    stNO_LENS[885].fEnergy := 29760.957445; stNO_LENS[885].fLow := 4.726807; stNO_LENS[885].fHigh := 9.548423;
    stNO_LENS[886].fEnergy := 29820.538922; stNO_LENS[886].fLow := 4.709276; stNO_LENS[886].fHigh := 9.507957;
    stNO_LENS[887].fEnergy := 29880.239680; stNO_LENS[887].fLow := 4.691804; stNO_LENS[887].fHigh := 9.467684;
    stNO_LENS[888].fEnergy := 29940.059960; stNO_LENS[888].fLow := 4.674389; stNO_LENS[888].fHigh := 9.427603;
    stNO_LENS[889].fEnergy := 30000.000000; stNO_LENS[889].fLow := 4.657032; stNO_LENS[889].fHigh := 9.387713;
    stNO_LENS[890].fEnergy := 30068.760232; stNO_LENS[890].fLow := 4.637235; stNO_LENS[890].fHigh := 9.342285;
    stNO_LENS[891].fEnergy := 30128.957930; stNO_LENS[891].fLow := 4.620001; stNO_LENS[891].fHigh := 9.302803;
    stNO_LENS[892].fEnergy := 30189.276144; stNO_LENS[892].fLow := 4.602825; stNO_LENS[892].fHigh := 9.263510;
    stNO_LENS[893].fEnergy := 30249.715115; stNO_LENS[893].fLow := 4.585705; stNO_LENS[893].fHigh := 9.224405;
    stNO_LENS[894].fEnergy := 30310.275085; stNO_LENS[894].fLow := 4.568643; stNO_LENS[894].fHigh := 9.185487;
    stNO_LENS[895].fEnergy := 30370.956297; stNO_LENS[895].fLow := 4.551636; stNO_LENS[895].fHigh := 9.146757;
    stNO_LENS[896].fEnergy := 30431.758992; stNO_LENS[896].fLow := 4.534686; stNO_LENS[896].fHigh := 9.108213;
    stNO_LENS[897].fEnergy := 30492.683414; stNO_LENS[897].fLow := 4.517791; stNO_LENS[897].fHigh := 9.069854;
    stNO_LENS[898].fEnergy := 30553.729807; stNO_LENS[898].fLow := 4.500952; stNO_LENS[898].fHigh := 9.031681;
    stNO_LENS[899].fEnergy := 30614.898414; stNO_LENS[899].fLow := 4.484169; stNO_LENS[899].fHigh := 8.993692;
    stNO_LENS[900].fEnergy := 30676.189482; stNO_LENS[900].fLow := 4.467441; stNO_LENS[900].fHigh := 8.955886;
    stNO_LENS[901].fEnergy := 30737.603254; stNO_LENS[901].fLow := 4.450767; stNO_LENS[901].fHigh := 8.918263;
    stNO_LENS[902].fEnergy := 30799.139977; stNO_LENS[902].fLow := 4.434149; stNO_LENS[902].fHigh := 8.880822;
    stNO_LENS[903].fEnergy := 30860.799896; stNO_LENS[903].fLow := 4.417585; stNO_LENS[903].fHigh := 8.843563;
    stNO_LENS[904].fEnergy := 30922.583259; stNO_LENS[904].fLow := 4.401076; stNO_LENS[904].fHigh := 8.806484;
    stNO_LENS[905].fEnergy := 30984.490312; stNO_LENS[905].fLow := 4.384620; stNO_LENS[905].fHigh := 8.769586;
    stNO_LENS[906].fEnergy := 31046.521303; stNO_LENS[906].fLow := 4.368218; stNO_LENS[906].fHigh := 8.732867;
    stNO_LENS[907].fEnergy := 31108.676480; stNO_LENS[907].fLow := 4.351870; stNO_LENS[907].fHigh := 8.696327;
    stNO_LENS[908].fEnergy := 31170.956091; stNO_LENS[908].fLow := 4.335576; stNO_LENS[908].fHigh := 8.659965;
    stNO_LENS[909].fEnergy := 31233.360387; stNO_LENS[909].fLow := 4.319334; stNO_LENS[909].fHigh := 8.623781;
    stNO_LENS[910].fEnergy := 31295.889616; stNO_LENS[910].fLow := 4.303146; stNO_LENS[910].fHigh := 8.587773;
    stNO_LENS[911].fEnergy := 31358.544029; stNO_LENS[911].fLow := 4.287010; stNO_LENS[911].fHigh := 8.551941;
    stNO_LENS[912].fEnergy := 31421.323876; stNO_LENS[912].fLow := 4.270927; stNO_LENS[912].fHigh := 8.516285;
    stNO_LENS[913].fEnergy := 31484.229408; stNO_LENS[913].fLow := 4.254897; stNO_LENS[913].fHigh := 8.480803;
    stNO_LENS[914].fEnergy := 31547.260878; stNO_LENS[914].fLow := 4.238918; stNO_LENS[914].fHigh := 8.445496;
    stNO_LENS[915].fEnergy := 31610.418536; stNO_LENS[915].fLow := 4.222991; stNO_LENS[915].fHigh := 8.410362;
    stNO_LENS[916].fEnergy := 31673.702636; stNO_LENS[916].fLow := 4.207116; stNO_LENS[916].fHigh := 8.375401;
    stNO_LENS[917].fEnergy := 31737.113431; stNO_LENS[917].fLow := 4.191293; stNO_LENS[917].fHigh := 8.340611;
    stNO_LENS[918].fEnergy := 31800.651174; stNO_LENS[918].fLow := 4.175521; stNO_LENS[918].fHigh := 8.305993;
    stNO_LENS[919].fEnergy := 31864.316120; stNO_LENS[919].fLow := 4.159799; stNO_LENS[919].fHigh := 8.271546;
    stNO_LENS[920].fEnergy := 31928.108524; stNO_LENS[920].fLow := 4.144129; stNO_LENS[920].fHigh := 8.237269;
    stNO_LENS[921].fEnergy := 31992.028640; stNO_LENS[921].fLow := 4.128510; stNO_LENS[921].fHigh := 8.203161;
    stNO_LENS[922].fEnergy := 32056.076724; stNO_LENS[922].fLow := 4.112940; stNO_LENS[922].fHigh := 8.169222;
    stNO_LENS[923].fEnergy := 32120.253032; stNO_LENS[923].fLow := 4.097421; stNO_LENS[923].fHigh := 8.135452;
    stNO_LENS[924].fEnergy := 32184.557822; stNO_LENS[924].fLow := 4.081953; stNO_LENS[924].fHigh := 8.101848;
    stNO_LENS[925].fEnergy := 32248.991349; stNO_LENS[925].fLow := 4.066534; stNO_LENS[925].fHigh := 8.068411;
    stNO_LENS[926].fEnergy := 32313.553873; stNO_LENS[926].fLow := 4.051164; stNO_LENS[926].fHigh := 8.035141;
    stNO_LENS[927].fEnergy := 32378.245651; stNO_LENS[927].fLow := 4.035844; stNO_LENS[927].fHigh := 8.002035;
    stNO_LENS[928].fEnergy := 32443.066942; stNO_LENS[928].fLow := 4.020574; stNO_LENS[928].fHigh := 7.969095;
    stNO_LENS[929].fEnergy := 32508.018005; stNO_LENS[929].fLow := 4.005352; stNO_LENS[929].fHigh := 7.936319;
    stNO_LENS[930].fEnergy := 32573.099101; stNO_LENS[930].fLow := 3.990180; stNO_LENS[930].fHigh := 7.903706;
    stNO_LENS[931].fEnergy := 32638.310488; stNO_LENS[931].fLow := 3.975056; stNO_LENS[931].fHigh := 7.871256;
    stNO_LENS[932].fEnergy := 32703.652430; stNO_LENS[932].fLow := 3.959980; stNO_LENS[932].fHigh := 7.838968;
    stNO_LENS[933].fEnergy := 32769.125185; stNO_LENS[933].fLow := 3.944953; stNO_LENS[933].fHigh := 7.806842;
    stNO_LENS[934].fEnergy := 32834.729018; stNO_LENS[934].fLow := 3.929974; stNO_LENS[934].fHigh := 7.774876;
    stNO_LENS[935].fEnergy := 32900.464189; stNO_LENS[935].fLow := 3.915043; stNO_LENS[935].fHigh := 7.743071;
    stNO_LENS[936].fEnergy := 32966.330962; stNO_LENS[936].fLow := 3.900159; stNO_LENS[936].fHigh := 7.711425;
    stNO_LENS[937].fEnergy := 33032.329601; stNO_LENS[937].fLow := 3.885323; stNO_LENS[937].fHigh := 7.679938;
    stNO_LENS[938].fEnergy := 33098.460369; stNO_LENS[938].fLow := 3.870535; stNO_LENS[938].fHigh := 7.648610;
    stNO_LENS[939].fEnergy := 33164.723530; stNO_LENS[939].fLow := 3.855793; stNO_LENS[939].fHigh := 7.617439;
    stNO_LENS[940].fEnergy := 33231.119351; stNO_LENS[940].fLow := 3.841099; stNO_LENS[940].fHigh := 7.586425;
    stNO_LENS[941].fEnergy := 33297.648096; stNO_LENS[941].fLow := 3.826451; stNO_LENS[941].fHigh := 7.555568;
    stNO_LENS[942].fEnergy := 33364.310032; stNO_LENS[942].fLow := 3.811850; stNO_LENS[942].fHigh := 7.524866;
    stNO_LENS[943].fEnergy := 33431.105426; stNO_LENS[943].fLow := 3.797296; stNO_LENS[943].fHigh := 7.494320;
    stNO_LENS[944].fEnergy := 33498.034543; stNO_LENS[944].fLow := 3.782787; stNO_LENS[944].fHigh := 7.463928;
    stNO_LENS[945].fEnergy := 33565.097653; stNO_LENS[945].fLow := 3.768325; stNO_LENS[945].fHigh := 7.433689;
    stNO_LENS[946].fEnergy := 33632.295023; stNO_LENS[946].fLow := 3.753909; stNO_LENS[946].fHigh := 7.389056;
    stNO_LENS[947].fEnergy := 33699.626923; stNO_LENS[947].fLow := 3.739538; stNO_LENS[947].fHigh := 7.389056;
    stNO_LENS[948].fEnergy := 33767.093621; stNO_LENS[948].fLow := 3.725213; stNO_LENS[948].fHigh := 7.320540;
    stNO_LENS[949].fEnergy := 33834.695387; stNO_LENS[949].fLow := 3.710933; stNO_LENS[949].fHigh := 7.130147;
    stNO_LENS[950].fEnergy := 33902.432493; stNO_LENS[950].fLow := 3.696699; stNO_LENS[950].fHigh := 6.944706;
    stNO_LENS[951].fEnergy := 33970.305208; stNO_LENS[951].fLow := 3.682509; stNO_LENS[951].fHigh := 6.764088;
    stNO_LENS[952].fEnergy := 34038.313804; stNO_LENS[952].fLow := 3.668365; stNO_LENS[952].fHigh := 6.588167;
    stNO_LENS[953].fEnergy := 34106.458554; stNO_LENS[953].fLow := 3.654265; stNO_LENS[953].fHigh := 6.416822;
    stNO_LENS[954].fEnergy := 34174.739729; stNO_LENS[954].fLow := 3.640209; stNO_LENS[954].fHigh := 6.249933;
    stNO_LENS[955].fEnergy := 34243.157604; stNO_LENS[955].fLow := 3.626198; stNO_LENS[955].fHigh := 6.087384;
    stNO_LENS[956].fEnergy := 34311.712451; stNO_LENS[956].fLow := 3.612231; stNO_LENS[956].fHigh := 5.929063;
    stNO_LENS[957].fEnergy := 34380.404545; stNO_LENS[957].fLow := 3.598308; stNO_LENS[957].fHigh := 5.774860;
    stNO_LENS[958].fEnergy := 34449.234161; stNO_LENS[958].fLow := 3.584429; stNO_LENS[958].fHigh := 5.624667;
    stNO_LENS[959].fEnergy := 34518.201574; stNO_LENS[959].fLow := 3.570593; stNO_LENS[959].fHigh := 5.478381;
    stNO_LENS[960].fEnergy := 34587.307059; stNO_LENS[960].fLow := 3.556802; stNO_LENS[960].fHigh := 5.335899;
    stNO_LENS[961].fEnergy := 34656.550894; stNO_LENS[961].fLow := 3.543053; stNO_LENS[961].fHigh := 5.197123;
    stNO_LENS[962].fEnergy := 34725.933355; stNO_LENS[962].fLow := 3.529348; stNO_LENS[962].fHigh := 5.061956;
    stNO_LENS[963].fEnergy := 34795.454720; stNO_LENS[963].fLow := 3.515685; stNO_LENS[963].fHigh := 4.930304;
    stNO_LENS[964].fEnergy := 34865.115267; stNO_LENS[964].fLow := 3.502066; stNO_LENS[964].fHigh := 4.802077;
    stNO_LENS[965].fEnergy := 34934.915274; stNO_LENS[965].fLow := 3.488489; stNO_LENS[965].fHigh := 4.677184;
    stNO_LENS[966].fEnergy := 35004.855021; stNO_LENS[966].fLow := 3.474955; stNO_LENS[966].fHigh := 4.555540;
    stNO_LENS[967].fEnergy := 35074.934788; stNO_LENS[967].fLow := 3.461463; stNO_LENS[967].fHigh := 4.437059;
    stNO_LENS[968].fEnergy := 35145.154854; stNO_LENS[968].fLow := 3.448013; stNO_LENS[968].fHigh := 4.321660;
    stNO_LENS[969].fEnergy := 35215.515501; stNO_LENS[969].fLow := 3.434605; stNO_LENS[969].fHigh := 4.209262;
    stNO_LENS[970].fEnergy := 35286.017010; stNO_LENS[970].fLow := 3.421240; stNO_LENS[970].fHigh := 4.099787;
    stNO_LENS[971].fEnergy := 35356.659663; stNO_LENS[971].fLow := 3.407916; stNO_LENS[971].fHigh := 3.993160;
    stNO_LENS[972].fEnergy := 35427.443743; stNO_LENS[972].fLow := 3.394634; stNO_LENS[972].fHigh := 3.889306;
    stNO_LENS[973].fEnergy := 35498.369532; stNO_LENS[973].fLow := 3.381393; stNO_LENS[973].fHigh := 3.788152;
    stNO_LENS[974].fEnergy := 35569.437315; stNO_LENS[974].fLow := 3.368193; stNO_LENS[974].fHigh := 3.689630;
    stNO_LENS[975].fEnergy := 35640.647376; stNO_LENS[975].fLow := 3.355035; stNO_LENS[975].fHigh := 3.593670;
    stNO_LENS[976].fEnergy := 35712.000000; stNO_LENS[976].fLow := 3.341917; stNO_LENS[976].fHigh := 3.500206;
    stNO_LENS[977].fEnergy := 35783.495472; stNO_LENS[977].fLow := 3.328841; stNO_LENS[977].fHigh := 3.409172;
    stNO_LENS[978].fEnergy := 35855.134077; stNO_LENS[978].fLow := 3.315805; stNO_LENS[978].fHigh := 3.320506;


    stLENS3_333[0].fEnergy := 9500.000000; stLENS3_333[0].fLow := 41.170000; stLENS3_333[0].fHigh := 10000.000000;
    stLENS3_333[1].fEnergy := 9518.120298; stLENS3_333[1].fLow := 40.979550; stLENS3_333[1].fHigh := 10000.000000;
    stLENS3_333[2].fEnergy := 9537.175588; stLENS3_333[2].fLow := 40.775094; stLENS3_333[2].fHigh := 10000.000000;
    stLENS3_333[3].fEnergy := 9556.269026; stLENS3_333[3].fLow := 40.572130; stLENS3_333[3].fHigh := 10000.000000;
    stLENS3_333[4].fEnergy := 9575.400690; stLENS3_333[4].fLow := 40.370644; stLENS3_333[4].fHigh := 10000.000000;
    stLENS3_333[5].fEnergy := 9594.570654; stLENS3_333[5].fLow := 40.170623; stLENS3_333[5].fHigh := 10000.000000;
    stLENS3_333[6].fEnergy := 9613.778998; stLENS3_333[6].fLow := 39.972052; stLENS3_333[6].fHigh := 10000.000000;
    stLENS3_333[7].fEnergy := 9633.025796; stLENS3_333[7].fLow := 39.774917; stLENS3_333[7].fHigh := 10000.000000;
    stLENS3_333[8].fEnergy := 9652.311127; stLENS3_333[8].fLow := 39.579205; stLENS3_333[8].fHigh := 10000.000000;
    stLENS3_333[9].fEnergy := 9671.635066; stLENS3_333[9].fLow := 39.384902; stLENS3_333[9].fHigh := 10000.000000;
    stLENS3_333[10].fEnergy := 9690.997693; stLENS3_333[10].fLow := 39.191996; stLENS3_333[10].fHigh := 10000.000000;
    stLENS3_333[11].fEnergy := 9710.399083; stLENS3_333[11].fLow := 39.000472; stLENS3_333[11].fHigh := 10000.000000;
    stLENS3_333[12].fEnergy := 9729.839315; stLENS3_333[12].fLow := 38.810318; stLENS3_333[12].fHigh := 10000.000000;
    stLENS3_333[13].fEnergy := 9749.318466; stLENS3_333[13].fLow := 38.621521; stLENS3_333[13].fHigh := 10000.000000;
    stLENS3_333[14].fEnergy := 9768.836615; stLENS3_333[14].fLow := 38.434067; stLENS3_333[14].fHigh := 10000.000000;
    stLENS3_333[15].fEnergy := 9788.393839; stLENS3_333[15].fLow := 38.247946; stLENS3_333[15].fHigh := 10000.000000;
    stLENS3_333[16].fEnergy := 9807.990216; stLENS3_333[16].fLow := 38.063143; stLENS3_333[16].fHigh := 10000.000000;
    stLENS3_333[17].fEnergy := 9827.625826; stLENS3_333[17].fLow := 37.879646; stLENS3_333[17].fHigh := 10000.000000;
    stLENS3_333[18].fEnergy := 9847.300746; stLENS3_333[18].fLow := 37.697444; stLENS3_333[18].fHigh := 10000.000000;
    stLENS3_333[19].fEnergy := 9867.015055; stLENS3_333[19].fLow := 37.516524; stLENS3_333[19].fHigh := 10000.000000;
    stLENS3_333[20].fEnergy := 9886.768832; stLENS3_333[20].fLow := 37.336875; stLENS3_333[20].fHigh := 10000.000000;
    stLENS3_333[21].fEnergy := 9906.562157; stLENS3_333[21].fLow := 37.158483; stLENS3_333[21].fHigh := 10000.000000;
    stLENS3_333[22].fEnergy := 9926.395107; stLENS3_333[22].fLow := 36.981339; stLENS3_333[22].fHigh := 10000.000000;
    stLENS3_333[23].fEnergy := 9946.267764; stLENS3_333[23].fLow := 36.805429; stLENS3_333[23].fHigh := 10000.000000;
    stLENS3_333[24].fEnergy := 9966.180205; stLENS3_333[24].fLow := 36.630742; stLENS3_333[24].fHigh := 10000.000000;
    stLENS3_333[25].fEnergy := 9986.132511; stLENS3_333[25].fLow := 36.457268; stLENS3_333[25].fHigh := 10000.000000;
    stLENS3_333[26].fEnergy := 10006.124762; stLENS3_333[26].fLow := 36.284994; stLENS3_333[26].fHigh := 10000.000000;
    stLENS3_333[27].fEnergy := 10026.157037; stLENS3_333[27].fLow := 36.113911; stLENS3_333[27].fHigh := 10000.000000;
    stLENS3_333[28].fEnergy := 10046.229416; stLENS3_333[28].fLow := 35.944006; stLENS3_333[28].fHigh := 10000.000000;
    stLENS3_333[29].fEnergy := 10066.341981; stLENS3_333[29].fLow := 35.775268; stLENS3_333[29].fHigh := 10000.000000;
    stLENS3_333[30].fEnergy := 10086.494811; stLENS3_333[30].fLow := 35.607688; stLENS3_333[30].fHigh := 10000.000000;
    stLENS3_333[31].fEnergy := 10106.687987; stLENS3_333[31].fLow := 35.441254; stLENS3_333[31].fHigh := 10000.000000;
    stLENS3_333[32].fEnergy := 10126.921590; stLENS3_333[32].fLow := 35.275956; stLENS3_333[32].fHigh := 10000.000000;
    stLENS3_333[33].fEnergy := 10147.195701; stLENS3_333[33].fLow := 35.111783; stLENS3_333[33].fHigh := 10000.000000;
    stLENS3_333[34].fEnergy := 10167.510400; stLENS3_333[34].fLow := 34.948725; stLENS3_333[34].fHigh := 10000.000000;
    stLENS3_333[35].fEnergy := 10187.865769; stLENS3_333[35].fLow := 34.786771; stLENS3_333[35].fHigh := 10000.000000;
    stLENS3_333[36].fEnergy := 10208.261890; stLENS3_333[36].fLow := 34.625913; stLENS3_333[36].fHigh := 10000.000000;
    stLENS3_333[37].fEnergy := 10228.698844; stLENS3_333[37].fLow := 34.466138; stLENS3_333[37].fHigh := 10000.000000;
    stLENS3_333[38].fEnergy := 10249.176713; stLENS3_333[38].fLow := 34.307439; stLENS3_333[38].fHigh := 10000.000000;
    stLENS3_333[39].fEnergy := 10269.695578; stLENS3_333[39].fLow := 34.149804; stLENS3_333[39].fHigh := 10000.000000;
    stLENS3_333[40].fEnergy := 10290.255523; stLENS3_333[40].fLow := 33.993224; stLENS3_333[40].fHigh := 10000.000000;
    stLENS3_333[41].fEnergy := 10310.856628; stLENS3_333[41].fLow := 33.837689; stLENS3_333[41].fHigh := 10000.000000;
    stLENS3_333[42].fEnergy := 10331.498977; stLENS3_333[42].fLow := 33.683191; stLENS3_333[42].fHigh := 10000.000000;
    stLENS3_333[43].fEnergy := 10352.182651; stLENS3_333[43].fLow := 33.529719; stLENS3_333[43].fHigh := 10000.000000;
    stLENS3_333[44].fEnergy := 10372.907735; stLENS3_333[44].fLow := 33.377264; stLENS3_333[44].fHigh := 10000.000000;
    stLENS3_333[45].fEnergy := 10393.674310; stLENS3_333[45].fLow := 33.225816; stLENS3_333[45].fHigh := 10000.000000;
    stLENS3_333[46].fEnergy := 10414.482460; stLENS3_333[46].fLow := 33.075368; stLENS3_333[46].fHigh := 10000.000000;
    stLENS3_333[47].fEnergy := 10435.332268; stLENS3_333[47].fLow := 32.925909; stLENS3_333[47].fHigh := 10000.000000;
    stLENS3_333[48].fEnergy := 10456.223817; stLENS3_333[48].fLow := 32.777431; stLENS3_333[48].fHigh := 10000.000000;
    stLENS3_333[49].fEnergy := 10477.157191; stLENS3_333[49].fLow := 32.629925; stLENS3_333[49].fHigh := 10000.000000;
    stLENS3_333[50].fEnergy := 10498.132473; stLENS3_333[50].fLow := 32.483382; stLENS3_333[50].fHigh := 10000.000000;
    stLENS3_333[51].fEnergy := 10519.149749; stLENS3_333[51].fLow := 32.337793; stLENS3_333[51].fHigh := 10000.000000;
    stLENS3_333[52].fEnergy := 10540.209100; stLENS3_333[52].fLow := 32.193150; stLENS3_333[52].fHigh := 10000.000000;
    stLENS3_333[53].fEnergy := 10561.310613; stLENS3_333[53].fLow := 32.049444; stLENS3_333[53].fHigh := 10000.000000;
    stLENS3_333[54].fEnergy := 10582.454371; stLENS3_333[54].fLow := 31.906667; stLENS3_333[54].fHigh := 10000.000000;
    stLENS3_333[55].fEnergy := 10603.640459; stLENS3_333[55].fLow := 31.764811; stLENS3_333[55].fHigh := 10000.000000;
    stLENS3_333[56].fEnergy := 10624.868961; stLENS3_333[56].fLow := 31.623866; stLENS3_333[56].fHigh := 10000.000000;
    stLENS3_333[57].fEnergy := 10646.139963; stLENS3_333[57].fLow := 31.483826; stLENS3_333[57].fHigh := 10000.000000;
    stLENS3_333[58].fEnergy := 10667.453549; stLENS3_333[58].fLow := 31.344682; stLENS3_333[58].fHigh := 10000.000000;
    stLENS3_333[59].fEnergy := 10688.809806; stLENS3_333[59].fLow := 31.206425; stLENS3_333[59].fHigh := 10000.000000;
    stLENS3_333[60].fEnergy := 10710.208817; stLENS3_333[60].fLow := 31.069049; stLENS3_333[60].fHigh := 10000.000000;
    stLENS3_333[61].fEnergy := 10731.650669; stLENS3_333[61].fLow := 30.932544; stLENS3_333[61].fHigh := 10000.000000;
    stLENS3_333[62].fEnergy := 10753.135448; stLENS3_333[62].fLow := 30.796904; stLENS3_333[62].fHigh := 10000.000000;
    stLENS3_333[63].fEnergy := 10774.663240; stLENS3_333[63].fLow := 30.662121; stLENS3_333[63].fHigh := 10000.000000;
    stLENS3_333[64].fEnergy := 10796.234130; stLENS3_333[64].fLow := 30.528187; stLENS3_333[64].fHigh := 10000.000000;
    stLENS3_333[65].fEnergy := 10817.848205; stLENS3_333[65].fLow := 30.395094; stLENS3_333[65].fHigh := 10000.000000;
    stLENS3_333[66].fEnergy := 10839.505552; stLENS3_333[66].fLow := 30.262835; stLENS3_333[66].fHigh := 10000.000000;
    stLENS3_333[67].fEnergy := 10861.206256; stLENS3_333[67].fLow := 30.131403; stLENS3_333[67].fHigh := 10000.000000;
    stLENS3_333[68].fEnergy := 10882.950406; stLENS3_333[68].fLow := 30.000790; stLENS3_333[68].fHigh := 10000.000000;
    stLENS3_333[69].fEnergy := 10904.738087; stLENS3_333[69].fLow := 29.870989; stLENS3_333[69].fHigh := 10000.000000;
    stLENS3_333[70].fEnergy := 10926.569387; stLENS3_333[70].fLow := 29.741992; stLENS3_333[70].fHigh := 10000.000000;
    stLENS3_333[71].fEnergy := 10948.444394; stLENS3_333[71].fLow := 29.613794; stLENS3_333[71].fHigh := 10000.000000;
    stLENS3_333[72].fEnergy := 10970.363194; stLENS3_333[72].fLow := 29.486386; stLENS3_333[72].fHigh := 10000.000000;
    stLENS3_333[73].fEnergy := 10992.325876; stLENS3_333[73].fLow := 29.359762; stLENS3_333[73].fHigh := 10000.000000;
    stLENS3_333[74].fEnergy := 11014.332527; stLENS3_333[74].fLow := 29.233914; stLENS3_333[74].fHigh := 10000.000000;
    stLENS3_333[75].fEnergy := 11036.383235; stLENS3_333[75].fLow := 29.108837; stLENS3_333[75].fHigh := 10000.000000;
    stLENS3_333[76].fEnergy := 11058.478089; stLENS3_333[76].fLow := 28.984523; stLENS3_333[76].fHigh := 10000.000000;
    stLENS3_333[77].fEnergy := 11080.617177; stLENS3_333[77].fLow := 28.860965; stLENS3_333[77].fHigh := 10000.000000;
    stLENS3_333[78].fEnergy := 11102.800587; stLENS3_333[78].fLow := 28.738157; stLENS3_333[78].fHigh := 10000.000000;
    stLENS3_333[79].fEnergy := 11125.028409; stLENS3_333[79].fLow := 28.616092; stLENS3_333[79].fHigh := 10000.000000;
    stLENS3_333[80].fEnergy := 11147.300731; stLENS3_333[80].fLow := 28.494764; stLENS3_333[80].fHigh := 2982.710527;
    stLENS3_333[81].fEnergy := 11169.617642; stLENS3_333[81].fLow := 28.374167; stLENS3_333[81].fHigh := 2131.025109;
    stLENS3_333[82].fEnergy := 11191.979231; stLENS3_333[82].fLow := 28.254293; stLENS3_333[82].fHigh := 1522.530589;
    stLENS3_333[83].fEnergy := 11214.385588; stLENS3_333[83].fLow := 28.135137; stLENS3_333[83].fHigh := 1087.786054;
    stLENS3_333[84].fEnergy := 11236.836803; stLENS3_333[84].fLow := 28.016692; stLENS3_333[84].fHigh := 921.367411;
    stLENS3_333[85].fEnergy := 11259.332966; stLENS3_333[85].fLow := 27.898953; stLENS3_333[85].fHigh := 828.581439;
    stLENS3_333[86].fEnergy := 11281.874165; stLENS3_333[86].fLow := 27.781912; stLENS3_333[86].fHigh := 747.775297;
    stLENS3_333[87].fEnergy := 11304.460492; stLENS3_333[87].fLow := 27.665564; stLENS3_333[87].fHigh := 677.236862;
    stLENS3_333[88].fEnergy := 11327.092037; stLENS3_333[88].fLow := 27.549904; stLENS3_333[88].fHigh := 615.522063;
    stLENS3_333[89].fEnergy := 11349.768891; stLENS3_333[89].fLow := 27.434924; stLENS3_333[89].fHigh := 561.410100;
    stLENS3_333[90].fEnergy := 11372.491143; stLENS3_333[90].fLow := 27.320619; stLENS3_333[90].fHigh := 513.866586;
    stLENS3_333[91].fEnergy := 11395.258886; stLENS3_333[91].fLow := 27.206983; stLENS3_333[91].fHigh := 472.013149;
    stLENS3_333[92].fEnergy := 11418.072209; stLENS3_333[92].fLow := 27.094011; stLENS3_333[92].fHigh := 435.102297;
    stLENS3_333[93].fEnergy := 11440.931205; stLENS3_333[93].fLow := 26.981697; stLENS3_333[93].fHigh := 402.496600;
    stLENS3_333[94].fEnergy := 11463.835964; stLENS3_333[94].fLow := 26.870034; stLENS3_333[94].fHigh := 373.651402;
    stLENS3_333[95].fEnergy := 11486.786579; stLENS3_333[95].fLow := 26.759018; stLENS3_333[95].fHigh := 348.100445;
    stLENS3_333[96].fEnergy := 11509.783141; stLENS3_333[96].fLow := 26.648642; stLENS3_333[96].fHigh := 325.443874;
    stLENS3_333[97].fEnergy := 11532.825743; stLENS3_333[97].fLow := 26.538902; stLENS3_333[97].fHigh := 311.096768;
    stLENS3_333[98].fEnergy := 11555.914475; stLENS3_333[98].fLow := 26.429792; stLENS3_333[98].fHigh := 302.082371;
    stLENS3_333[99].fEnergy := 11579.049431; stLENS3_333[99].fLow := 26.321306; stLENS3_333[99].fHigh := 293.329178;
    stLENS3_333[100].fEnergy := 11602.230704; stLENS3_333[100].fLow := 26.213438; stLENS3_333[100].fHigh := 284.829619;
    stLENS3_333[101].fEnergy := 11625.458385; stLENS3_333[101].fLow := 26.106185; stLENS3_333[101].fHigh := 276.576344;
    stLENS3_333[102].fEnergy := 11648.732568; stLENS3_333[102].fLow := 25.999540; stLENS3_333[102].fHigh := 268.562218;
    stLENS3_333[103].fEnergy := 11672.053346; stLENS3_333[103].fLow := 25.893498; stLENS3_333[103].fHigh := 260.780310;
    stLENS3_333[104].fEnergy := 11695.420813; stLENS3_333[104].fLow := 25.788054; stLENS3_333[104].fHigh := 253.223893;
    stLENS3_333[105].fEnergy := 11718.835061; stLENS3_333[105].fLow := 25.683204; stLENS3_333[105].fHigh := 245.886432;
    stLENS3_333[106].fEnergy := 11742.296184; stLENS3_333[106].fLow := 25.578941; stLENS3_333[106].fHigh := 238.761582;
    stLENS3_333[107].fEnergy := 11765.804277; stLENS3_333[107].fLow := 25.475261; stLENS3_333[107].fHigh := 231.843183;
    stLENS3_333[108].fEnergy := 11789.359433; stLENS3_333[108].fLow := 25.372158; stLENS3_333[108].fHigh := 225.125253;
    stLENS3_333[109].fEnergy := 11812.961746; stLENS3_333[109].fLow := 25.269629; stLENS3_333[109].fHigh := 218.601983;
    stLENS3_333[110].fEnergy := 11836.611311; stLENS3_333[110].fLow := 25.167668; stLENS3_333[110].fHigh := 212.267732;
    stLENS3_333[111].fEnergy := 11860.308223; stLENS3_333[111].fLow := 25.066270; stLENS3_333[111].fHigh := 206.117024;
    stLENS3_333[112].fEnergy := 11884.052576; stLENS3_333[112].fLow := 24.965430; stLENS3_333[112].fHigh := 200.144540;
    stLENS3_333[113].fEnergy := 11907.844465; stLENS3_333[113].fLow := 24.865144; stLENS3_333[113].fHigh := 194.345115;
    stLENS3_333[114].fEnergy := 11931.683985; stLENS3_333[114].fLow := 24.765408; stLENS3_333[114].fHigh := 188.713736;
    stLENS3_333[115].fEnergy := 11955.571233; stLENS3_333[115].fLow := 24.666215; stLENS3_333[115].fHigh := 183.245533;
    stLENS3_333[116].fEnergy := 11979.506302; stLENS3_333[116].fLow := 24.567563; stLENS3_333[116].fHigh := 177.935777;
    stLENS3_333[117].fEnergy := 12003.489290; stLENS3_333[117].fLow := 24.469445; stLENS3_333[117].fHigh := 175.087873;
    stLENS3_333[118].fEnergy := 12027.520291; stLENS3_333[118].fLow := 24.371858; stLENS3_333[118].fHigh := 172.351551;
    stLENS3_333[119].fEnergy := 12051.599403; stLENS3_333[119].fLow := 24.274798; stLENS3_333[119].fHigh := 169.675793;
    stLENS3_333[120].fEnergy := 12075.726721; stLENS3_333[120].fLow := 24.178259; stLENS3_333[120].fHigh := 167.059103;
    stLENS3_333[121].fEnergy := 12099.902342; stLENS3_333[121].fLow := 24.082237; stLENS3_333[121].fHigh := 164.500023;
    stLENS3_333[122].fEnergy := 12124.126363; stLENS3_333[122].fLow := 23.986728; stLENS3_333[122].fHigh := 161.997140;
    stLENS3_333[123].fEnergy := 12148.398880; stLENS3_333[123].fLow := 23.891729; stLENS3_333[123].fHigh := 159.549076;
    stLENS3_333[124].fEnergy := 12172.719991; stLENS3_333[124].fLow := 23.797233; stLENS3_333[124].fHigh := 157.154493;
    stLENS3_333[125].fEnergy := 12197.089792; stLENS3_333[125].fLow := 23.703238; stLENS3_333[125].fHigh := 154.812091;
    stLENS3_333[126].fEnergy := 12221.508382; stLENS3_333[126].fLow := 23.609738; stLENS3_333[126].fHigh := 152.520603;
    stLENS3_333[127].fEnergy := 12245.975858; stLENS3_333[127].fLow := 23.516731; stLENS3_333[127].fHigh := 150.278798;
    stLENS3_333[128].fEnergy := 12270.492318; stLENS3_333[128].fLow := 23.424211; stLENS3_333[128].fHigh := 148.085480;
    stLENS3_333[129].fEnergy := 12295.057860; stLENS3_333[129].fLow := 23.332174; stLENS3_333[129].fHigh := 145.939483;
    stLENS3_333[130].fEnergy := 12319.672583; stLENS3_333[130].fLow := 23.240618; stLENS3_333[130].fHigh := 143.839675;
    stLENS3_333[131].fEnergy := 12344.336584; stLENS3_333[131].fLow := 23.149536; stLENS3_333[131].fHigh := 141.784954;
    stLENS3_333[132].fEnergy := 12369.049962; stLENS3_333[132].fLow := 23.058927; stLENS3_333[132].fHigh := 139.774248;
    stLENS3_333[133].fEnergy := 12393.812816; stLENS3_333[133].fLow := 22.968785; stLENS3_333[133].fHigh := 137.806513;
    stLENS3_333[134].fEnergy := 12418.625246; stLENS3_333[134].fLow := 22.879106; stLENS3_333[134].fHigh := 135.880736;
    stLENS3_333[135].fEnergy := 12443.487350; stLENS3_333[135].fLow := 22.789888; stLENS3_333[135].fHigh := 133.995927;
    stLENS3_333[136].fEnergy := 12468.399229; stLENS3_333[136].fLow := 22.701126; stLENS3_333[136].fHigh := 132.151126;
    stLENS3_333[137].fEnergy := 12493.360981; stLENS3_333[137].fLow := 22.612816; stLENS3_333[137].fHigh := 130.345398;
    stLENS3_333[138].fEnergy := 12518.372706; stLENS3_333[138].fLow := 22.524954; stLENS3_333[138].fHigh := 128.577832;
    stLENS3_333[139].fEnergy := 12543.434505; stLENS3_333[139].fLow := 22.437538; stLENS3_333[139].fHigh := 126.847543;
    stLENS3_333[140].fEnergy := 12568.546477; stLENS3_333[140].fLow := 22.350562; stLENS3_333[140].fHigh := 125.153669;
    stLENS3_333[141].fEnergy := 12593.708724; stLENS3_333[141].fLow := 22.264024; stLENS3_333[141].fHigh := 123.495369;
    stLENS3_333[142].fEnergy := 12618.921346; stLENS3_333[142].fLow := 22.177920; stLENS3_333[142].fHigh := 121.871828;
    stLENS3_333[143].fEnergy := 12644.184443; stLENS3_333[143].fLow := 22.092246; stLENS3_333[143].fHigh := 120.282249;
    stLENS3_333[144].fEnergy := 12669.498117; stLENS3_333[144].fLow := 22.006998; stLENS3_333[144].fHigh := 118.725859;
    stLENS3_333[145].fEnergy := 12694.862470; stLENS3_333[145].fLow := 21.922174; stLENS3_333[145].fHigh := 117.201902;
    stLENS3_333[146].fEnergy := 12720.277601; stLENS3_333[146].fLow := 21.837770; stLENS3_333[146].fHigh := 115.709646;
    stLENS3_333[147].fEnergy := 12745.743614; stLENS3_333[147].fLow := 21.753781; stLENS3_333[147].fHigh := 114.248376;
    stLENS3_333[148].fEnergy := 12771.260610; stLENS3_333[148].fLow := 21.670206; stLENS3_333[148].fHigh := 112.817395;
    stLENS3_333[149].fEnergy := 12796.828690; stLENS3_333[149].fLow := 21.587040; stLENS3_333[149].fHigh := 111.416026;
    stLENS3_333[150].fEnergy := 12822.447958; stLENS3_333[150].fLow := 21.504280; stLENS3_333[150].fHigh := 110.043608;
    stLENS3_333[151].fEnergy := 12848.118516; stLENS3_333[151].fLow := 21.421923; stLENS3_333[151].fHigh := 108.699499;
    stLENS3_333[152].fEnergy := 12873.840467; stLENS3_333[152].fLow := 21.339965; stLENS3_333[152].fHigh := 107.383073;
    stLENS3_333[153].fEnergy := 12899.613913; stLENS3_333[153].fLow := 21.258403; stLENS3_333[153].fHigh := 106.093720;
    stLENS3_333[154].fEnergy := 12925.438957; stLENS3_333[154].fLow := 21.177235; stLENS3_333[154].fHigh := 104.830846;
    stLENS3_333[155].fEnergy := 12951.315703; stLENS3_333[155].fLow := 21.096456; stLENS3_333[155].fHigh := 103.593872;
    stLENS3_333[156].fEnergy := 12977.244254; stLENS3_333[156].fLow := 21.016063; stLENS3_333[156].fHigh := 102.382235;
    stLENS3_333[157].fEnergy := 13003.224714; stLENS3_333[157].fLow := 20.936054; stLENS3_333[157].fHigh := 101.195386;
    stLENS3_333[158].fEnergy := 13029.257188; stLENS3_333[158].fLow := 20.856425; stLENS3_333[158].fHigh := 100.021216;
    stLENS3_333[159].fEnergy := 13055.341778; stLENS3_333[159].fLow := 20.777173; stLENS3_333[159].fHigh := 99.279602;
    stLENS3_333[160].fEnergy := 13081.478590; stLENS3_333[160].fLow := 20.698295; stLENS3_333[160].fHigh := 98.543487;
    stLENS3_333[161].fEnergy := 13107.667727; stLENS3_333[161].fLow := 20.619789; stLENS3_333[161].fHigh := 97.812830;
    stLENS3_333[162].fEnergy := 13133.909296; stLENS3_333[162].fLow := 20.541650; stLENS3_333[162].fHigh := 97.087590;
    stLENS3_333[163].fEnergy := 13160.203399; stLENS3_333[163].fLow := 20.463876; stLENS3_333[163].fHigh := 96.367728;
    stLENS3_333[164].fEnergy := 13186.550144; stLENS3_333[164].fLow := 20.386465; stLENS3_333[164].fHigh := 95.653203;
    stLENS3_333[165].fEnergy := 13212.949635; stLENS3_333[165].fLow := 20.309412; stLENS3_333[165].fHigh := 94.943976;
    stLENS3_333[166].fEnergy := 13239.401978; stLENS3_333[166].fLow := 20.232716; stLENS3_333[166].fHigh := 94.240008;
    stLENS3_333[167].fEnergy := 13265.907278; stLENS3_333[167].fLow := 20.156373; stLENS3_333[167].fHigh := 93.541259;
    stLENS3_333[168].fEnergy := 13292.465642; stLENS3_333[168].fLow := 20.080380; stLENS3_333[168].fHigh := 92.847691;
    stLENS3_333[169].fEnergy := 13319.077176; stLENS3_333[169].fLow := 20.004736; stLENS3_333[169].fHigh := 92.159266;
    stLENS3_333[170].fEnergy := 13345.741987; stLENS3_333[170].fLow := 19.929436; stLENS3_333[170].fHigh := 91.475945;
    stLENS3_333[171].fEnergy := 13372.460180; stLENS3_333[171].fLow := 19.854478; stLENS3_333[171].fHigh := 90.797691;
    stLENS3_333[172].fEnergy := 13399.231863; stLENS3_333[172].fLow := 19.779859; stLENS3_333[172].fHigh := 90.124465;
    stLENS3_333[173].fEnergy := 13426.057143; stLENS3_333[173].fLow := 19.705577; stLENS3_333[173].fHigh := 89.456231;
    stLENS3_333[174].fEnergy := 13452.936127; stLENS3_333[174].fLow := 19.631630; stLENS3_333[174].fHigh := 88.792952;
    stLENS3_333[175].fEnergy := 13479.868924; stLENS3_333[175].fLow := 19.558013; stLENS3_333[175].fHigh := 88.134591;
    stLENS3_333[176].fEnergy := 13506.855639; stLENS3_333[176].fLow := 19.484725; stLENS3_333[176].fHigh := 87.481111;
    stLENS3_333[177].fEnergy := 13533.896382; stLENS3_333[177].fLow := 19.411762; stLENS3_333[177].fHigh := 86.832477;
    stLENS3_333[178].fEnergy := 13560.991261; stLENS3_333[178].fLow := 19.339123; stLENS3_333[178].fHigh := 86.188652;
    stLENS3_333[179].fEnergy := 13588.140383; stLENS3_333[179].fLow := 19.266805; stLENS3_333[179].fHigh := 85.549600;
    stLENS3_333[180].fEnergy := 13615.343858; stLENS3_333[180].fLow := 19.194805; stLENS3_333[180].fHigh := 84.915287;
    stLENS3_333[181].fEnergy := 13642.601795; stLENS3_333[181].fLow := 19.123121; stLENS3_333[181].fHigh := 84.285677;
    stLENS3_333[182].fEnergy := 13669.914302; stLENS3_333[182].fLow := 19.051750; stLENS3_333[182].fHigh := 83.660736;
    stLENS3_333[183].fEnergy := 13697.281489; stLENS3_333[183].fLow := 18.980689; stLENS3_333[183].fHigh := 83.040428;
    stLENS3_333[184].fEnergy := 13724.703465; stLENS3_333[184].fLow := 18.909937; stLENS3_333[184].fHigh := 82.424719;
    stLENS3_333[185].fEnergy := 13752.180339; stLENS3_333[185].fLow := 18.839491; stLENS3_333[185].fHigh := 81.813575;
    stLENS3_333[186].fEnergy := 13779.712223; stLENS3_333[186].fLow := 18.769347; stLENS3_333[186].fHigh := 81.206963;
    stLENS3_333[187].fEnergy := 13807.299225; stLENS3_333[187].fLow := 18.699505; stLENS3_333[187].fHigh := 80.604849;
    stLENS3_333[188].fEnergy := 13834.941456; stLENS3_333[188].fLow := 18.629961; stLENS3_333[188].fHigh := 80.007199;
    stLENS3_333[189].fEnergy := 13862.639028; stLENS3_333[189].fLow := 18.560714; stLENS3_333[189].fHigh := 79.413980;
    stLENS3_333[190].fEnergy := 13890.392049; stLENS3_333[190].fLow := 18.491760; stLENS3_333[190].fHigh := 78.825160;
    stLENS3_333[191].fEnergy := 13918.200633; stLENS3_333[191].fLow := 18.423098; stLENS3_333[191].fHigh := 78.240706;
    stLENS3_333[192].fEnergy := 13946.064889; stLENS3_333[192].fLow := 18.354725; stLENS3_333[192].fHigh := 77.660585;
    stLENS3_333[193].fEnergy := 13973.984929; stLENS3_333[193].fLow := 18.286639; stLENS3_333[193].fHigh := 77.084766;
    stLENS3_333[194].fEnergy := 14001.960866; stLENS3_333[194].fLow := 18.218837; stLENS3_333[194].fHigh := 76.513215;
    stLENS3_333[195].fEnergy := 14029.992810; stLENS3_333[195].fLow := 18.151318; stLENS3_333[195].fHigh := 75.945903;
    stLENS3_333[196].fEnergy := 14058.080875; stLENS3_333[196].fLow := 18.084080; stLENS3_333[196].fHigh := 75.382797;
    stLENS3_333[197].fEnergy := 14086.225171; stLENS3_333[197].fLow := 18.017119; stLENS3_333[197].fHigh := 74.823867;
    stLENS3_333[198].fEnergy := 14114.425813; stLENS3_333[198].fLow := 17.950435; stLENS3_333[198].fHigh := 74.269080;
    stLENS3_333[199].fEnergy := 14142.682912; stLENS3_333[199].fLow := 17.884024; stLENS3_333[199].fHigh := 73.718407;
    stLENS3_333[200].fEnergy := 14170.996582; stLENS3_333[200].fLow := 17.817885; stLENS3_333[200].fHigh := 73.171817;
    stLENS3_333[201].fEnergy := 14199.366936; stLENS3_333[201].fLow := 17.752015; stLENS3_333[201].fHigh := 72.629280;
    stLENS3_333[202].fEnergy := 14227.794088; stLENS3_333[202].fLow := 17.686412; stLENS3_333[202].fHigh := 72.090765;
    stLENS3_333[203].fEnergy := 14256.278151; stLENS3_333[203].fLow := 17.621075; stLENS3_333[203].fHigh := 71.556244;
    stLENS3_333[204].fEnergy := 14284.819238; stLENS3_333[204].fLow := 17.556001; stLENS3_333[204].fHigh := 71.025685;
    stLENS3_333[205].fEnergy := 14313.417466; stLENS3_333[205].fLow := 17.491189; stLENS3_333[205].fHigh := 70.499061;
    stLENS3_333[206].fEnergy := 14342.072946; stLENS3_333[206].fLow := 17.426635; stLENS3_333[206].fHigh := 69.976341;
    stLENS3_333[207].fEnergy := 14370.785796; stLENS3_333[207].fLow := 17.362339; stLENS3_333[207].fHigh := 69.457497;
    stLENS3_333[208].fEnergy := 14399.556128; stLENS3_333[208].fLow := 17.298298; stLENS3_333[208].fHigh := 68.942499;
    stLENS3_333[209].fEnergy := 14428.384059; stLENS3_333[209].fLow := 17.234511; stLENS3_333[209].fHigh := 68.431321;
    stLENS3_333[210].fEnergy := 14457.269703; stLENS3_333[210].fLow := 17.170974; stLENS3_333[210].fHigh := 67.923932;
    stLENS3_333[211].fEnergy := 14486.213176; stLENS3_333[211].fLow := 17.107687; stLENS3_333[211].fHigh := 67.420306;
    stLENS3_333[212].fEnergy := 14515.214594; stLENS3_333[212].fLow := 17.044647; stLENS3_333[212].fHigh := 66.920413;
    stLENS3_333[213].fEnergy := 14544.274073; stLENS3_333[213].fLow := 16.981853; stLENS3_333[213].fHigh := 66.424228;
    stLENS3_333[214].fEnergy := 14573.391729; stLENS3_333[214].fLow := 16.919303; stLENS3_333[214].fHigh := 65.931721;
    stLENS3_333[215].fEnergy := 14602.567679; stLENS3_333[215].fLow := 16.856995; stLENS3_333[215].fHigh := 65.442866;
    stLENS3_333[216].fEnergy := 14631.802039; stLENS3_333[216].fLow := 16.794926; stLENS3_333[216].fHigh := 64.957635;
    stLENS3_333[217].fEnergy := 14661.094926; stLENS3_333[217].fLow := 16.733096; stLENS3_333[217].fHigh := 64.476003;
    stLENS3_333[218].fEnergy := 14690.446458; stLENS3_333[218].fLow := 16.671502; stLENS3_333[218].fHigh := 63.997941;
    stLENS3_333[219].fEnergy := 14719.856751; stLENS3_333[219].fLow := 16.610142; stLENS3_333[219].fHigh := 63.523424;
    stLENS3_333[220].fEnergy := 14749.325924; stLENS3_333[220].fLow := 16.549016; stLENS3_333[220].fHigh := 63.052426;
    stLENS3_333[221].fEnergy := 14778.854094; stLENS3_333[221].fLow := 16.488120; stLENS3_333[221].fHigh := 62.584919;
    stLENS3_333[222].fEnergy := 14808.441380; stLENS3_333[222].fLow := 16.427453; stLENS3_333[222].fHigh := 62.120879;
    stLENS3_333[223].fEnergy := 14838.087899; stLENS3_333[223].fLow := 16.367015; stLENS3_333[223].fHigh := 61.660280;
    stLENS3_333[224].fEnergy := 14867.793771; stLENS3_333[224].fLow := 16.306802; stLENS3_333[224].fHigh := 61.203096;
    stLENS3_333[225].fEnergy := 14897.559114; stLENS3_333[225].fLow := 16.246813; stLENS3_333[225].fHigh := 60.749301;
    stLENS3_333[226].fEnergy := 14927.384047; stLENS3_333[226].fLow := 16.187046; stLENS3_333[226].fHigh := 60.298872;
    stLENS3_333[227].fEnergy := 14957.268690; stLENS3_333[227].fLow := 16.127501; stLENS3_333[227].fHigh := 59.851782;
    stLENS3_333[228].fEnergy := 14987.213162; stLENS3_333[228].fLow := 16.068174; stLENS3_333[228].fHigh := 59.408007;
    stLENS3_333[229].fEnergy := 15017.217582; stLENS3_333[229].fLow := 16.009065; stLENS3_333[229].fHigh := 58.967522;
    stLENS3_333[230].fEnergy := 15047.282072; stLENS3_333[230].fLow := 15.950172; stLENS3_333[230].fHigh := 58.530304;
    stLENS3_333[231].fEnergy := 15077.406751; stLENS3_333[231].fLow := 15.891493; stLENS3_333[231].fHigh := 58.096327;
    stLENS3_333[232].fEnergy := 15107.591739; stLENS3_333[232].fLow := 15.833027; stLENS3_333[232].fHigh := 57.665568;
    stLENS3_333[233].fEnergy := 15137.837158; stLENS3_333[233].fLow := 15.774772; stLENS3_333[233].fHigh := 57.238003;
    stLENS3_333[234].fEnergy := 15168.143128; stLENS3_333[234].fLow := 15.716726; stLENS3_333[234].fHigh := 56.813608;
    stLENS3_333[235].fEnergy := 15198.509771; stLENS3_333[235].fLow := 15.658889; stLENS3_333[235].fHigh := 56.392359;
    stLENS3_333[236].fEnergy := 15228.937208; stLENS3_333[236].fLow := 15.601258; stLENS3_333[236].fHigh := 55.868600;
    stLENS3_333[237].fEnergy := 15259.425560; stLENS3_333[237].fLow := 15.543832; stLENS3_333[237].fHigh := 55.557880;
    stLENS3_333[238].fEnergy := 15289.974951; stLENS3_333[238].fLow := 15.486609; stLENS3_333[238].fHigh := 55.249113;
    stLENS3_333[239].fEnergy := 15320.585501; stLENS3_333[239].fLow := 15.429588; stLENS3_333[239].fHigh := 54.942284;
    stLENS3_333[240].fEnergy := 15351.257334; stLENS3_333[240].fLow := 15.372768; stLENS3_333[240].fHigh := 54.637382;
    stLENS3_333[241].fEnergy := 15381.990571; stLENS3_333[241].fLow := 15.316147; stLENS3_333[241].fHigh := 54.334393;
    stLENS3_333[242].fEnergy := 15412.785337; stLENS3_333[242].fLow := 15.259724; stLENS3_333[242].fHigh := 54.033303;
    stLENS3_333[243].fEnergy := 15443.641754; stLENS3_333[243].fLow := 15.203496; stLENS3_333[243].fHigh := 53.734101;
    stLENS3_333[244].fEnergy := 15474.559945; stLENS3_333[244].fLow := 15.147464; stLENS3_333[244].fHigh := 53.436772;
    stLENS3_333[245].fEnergy := 15505.540035; stLENS3_333[245].fLow := 15.091624; stLENS3_333[245].fHigh := 53.141304;
    stLENS3_333[246].fEnergy := 15536.582147; stLENS3_333[246].fLow := 15.035977; stLENS3_333[246].fHigh := 52.847685;
    stLENS3_333[247].fEnergy := 15567.686405; stLENS3_333[247].fLow := 14.980520; stLENS3_333[247].fHigh := 52.555902;
    stLENS3_333[248].fEnergy := 15598.852934; stLENS3_333[248].fLow := 14.925252; stLENS3_333[248].fHigh := 52.265942;
    stLENS3_333[249].fEnergy := 15630.081858; stLENS3_333[249].fLow := 14.870173; stLENS3_333[249].fHigh := 51.977793;
    stLENS3_333[250].fEnergy := 15661.373303; stLENS3_333[250].fLow := 14.815279; stLENS3_333[250].fHigh := 51.691443;
    stLENS3_333[251].fEnergy := 15692.727393; stLENS3_333[251].fLow := 14.760571; stLENS3_333[251].fHigh := 51.406879;
    stLENS3_333[252].fEnergy := 15724.144254; stLENS3_333[252].fLow := 14.706047; stLENS3_333[252].fHigh := 51.124089;
    stLENS3_333[253].fEnergy := 15755.624012; stLENS3_333[253].fLow := 14.651705; stLENS3_333[253].fHigh := 50.843062;
    stLENS3_333[254].fEnergy := 15787.166792; stLENS3_333[254].fLow := 14.597544; stLENS3_333[254].fHigh := 50.563785;
    stLENS3_333[255].fEnergy := 15818.772721; stLENS3_333[255].fLow := 14.543564; stLENS3_333[255].fHigh := 50.286246;
    stLENS3_333[256].fEnergy := 15850.441925; stLENS3_333[256].fLow := 14.489762; stLENS3_333[256].fHigh := 50.010434;
    stLENS3_333[257].fEnergy := 15882.174531; stLENS3_333[257].fLow := 14.436138; stLENS3_333[257].fHigh := 49.736337;
    stLENS3_333[258].fEnergy := 15913.970666; stLENS3_333[258].fLow := 14.382690; stLENS3_333[258].fHigh := 49.463943;
    stLENS3_333[259].fEnergy := 15945.830456; stLENS3_333[259].fLow := 14.329416; stLENS3_333[259].fHigh := 49.193241;
    stLENS3_333[260].fEnergy := 15977.754030; stLENS3_333[260].fLow := 14.276317; stLENS3_333[260].fHigh := 48.924219;
    stLENS3_333[261].fEnergy := 16009.741515; stLENS3_333[261].fLow := 14.223390; stLENS3_333[261].fHigh := 48.656866;
    stLENS3_333[262].fEnergy := 16041.793039; stLENS3_333[262].fLow := 14.170635; stLENS3_333[262].fHigh := 48.391171;
    stLENS3_333[263].fEnergy := 16073.908730; stLENS3_333[263].fLow := 14.118050; stLENS3_333[263].fHigh := 48.127122;
    stLENS3_333[264].fEnergy := 16106.088717; stLENS3_333[264].fLow := 14.065634; stLENS3_333[264].fHigh := 47.864708;
    stLENS3_333[265].fEnergy := 16138.333128; stLENS3_333[265].fLow := 14.013385; stLENS3_333[265].fHigh := 47.603919;
    stLENS3_333[266].fEnergy := 16170.642092; stLENS3_333[266].fLow := 13.961304; stLENS3_333[266].fHigh := 47.344743;
    stLENS3_333[267].fEnergy := 16203.015739; stLENS3_333[267].fLow := 13.909388; stLENS3_333[267].fHigh := 47.087169;
    stLENS3_333[268].fEnergy := 16235.454198; stLENS3_333[268].fLow := 13.857636; stLENS3_333[268].fHigh := 46.831187;
    stLENS3_333[269].fEnergy := 16267.957599; stLENS3_333[269].fLow := 13.806048; stLENS3_333[269].fHigh := 46.576786;
    stLENS3_333[270].fEnergy := 16300.526072; stLENS3_333[270].fLow := 13.754622; stLENS3_333[270].fHigh := 46.323955;
    stLENS3_333[271].fEnergy := 16333.159747; stLENS3_333[271].fLow := 13.703357; stLENS3_333[271].fHigh := 46.072684;
    stLENS3_333[272].fEnergy := 16365.858755; stLENS3_333[272].fLow := 13.652252; stLENS3_333[272].fHigh := 45.822962;
    stLENS3_333[273].fEnergy := 16398.623226; stLENS3_333[273].fLow := 13.601307; stLENS3_333[273].fHigh := 45.574778;
    stLENS3_333[274].fEnergy := 16431.453291; stLENS3_333[274].fLow := 13.550519; stLENS3_333[274].fHigh := 45.328123;
    stLENS3_333[275].fEnergy := 16464.349083; stLENS3_333[275].fLow := 13.499888; stLENS3_333[275].fHigh := 45.082986;
    stLENS3_333[276].fEnergy := 16497.310732; stLENS3_333[276].fLow := 13.449413; stLENS3_333[276].fHigh := 44.839357;
    stLENS3_333[277].fEnergy := 16530.338370; stLENS3_333[277].fLow := 13.399093; stLENS3_333[277].fHigh := 44.597226;
    stLENS3_333[278].fEnergy := 16563.432129; stLENS3_333[278].fLow := 13.348927; stLENS3_333[278].fHigh := 44.356583;
    stLENS3_333[279].fEnergy := 16596.592142; stLENS3_333[279].fLow := 13.298913; stLENS3_333[279].fHigh := 44.117417;
    stLENS3_333[280].fEnergy := 16629.818542; stLENS3_333[280].fLow := 13.249051; stLENS3_333[280].fHigh := 43.879719;
    stLENS3_333[281].fEnergy := 16663.111461; stLENS3_333[281].fLow := 13.199340; stLENS3_333[281].fHigh := 43.643479;
    stLENS3_333[282].fEnergy := 16696.471032; stLENS3_333[282].fLow := 13.149779; stLENS3_333[282].fHigh := 43.408688;
    stLENS3_333[283].fEnergy := 16729.897390; stLENS3_333[283].fLow := 13.100367; stLENS3_333[283].fHigh := 43.175335;
    stLENS3_333[284].fEnergy := 16763.390666; stLENS3_333[284].fLow := 13.051103; stLENS3_333[284].fHigh := 42.943411;
    stLENS3_333[285].fEnergy := 16796.950997; stLENS3_333[285].fLow := 13.001986; stLENS3_333[285].fHigh := 42.712906;
    stLENS3_333[286].fEnergy := 16830.578515; stLENS3_333[286].fLow := 12.953015; stLENS3_333[286].fHigh := 42.483812;
    stLENS3_333[287].fEnergy := 16864.273356; stLENS3_333[287].fLow := 12.904189; stLENS3_333[287].fHigh := 42.256117;
    stLENS3_333[288].fEnergy := 16898.035654; stLENS3_333[288].fLow := 12.855507; stLENS3_333[288].fHigh := 42.029814;
    stLENS3_333[289].fEnergy := 16931.865544; stLENS3_333[289].fLow := 12.806969; stLENS3_333[289].fHigh := 41.804893;
    stLENS3_333[290].fEnergy := 16965.763161; stLENS3_333[290].fLow := 12.758573; stLENS3_333[290].fHigh := 41.581344;
    stLENS3_333[291].fEnergy := 16999.728641; stLENS3_333[291].fLow := 12.710319; stLENS3_333[291].fHigh := 41.359159;
    stLENS3_333[292].fEnergy := 17033.762121; stLENS3_333[292].fLow := 12.662205; stLENS3_333[292].fHigh := 41.138328;
    stLENS3_333[293].fEnergy := 17067.863735; stLENS3_333[293].fLow := 12.614231; stLENS3_333[293].fHigh := 40.918843;
    stLENS3_333[294].fEnergy := 17102.033621; stLENS3_333[294].fLow := 12.566396; stLENS3_333[294].fHigh := 40.700694;
    stLENS3_333[295].fEnergy := 17136.271915; stLENS3_333[295].fLow := 12.518699; stLENS3_333[295].fHigh := 40.483873;
    stLENS3_333[296].fEnergy := 17170.578755; stLENS3_333[296].fLow := 12.471139; stLENS3_333[296].fHigh := 40.268370;
    stLENS3_333[297].fEnergy := 17204.954276; stLENS3_333[297].fLow := 12.423716; stLENS3_333[297].fHigh := 40.054177;
    stLENS3_333[298].fEnergy := 17239.398618; stLENS3_333[298].fLow := 12.376428; stLENS3_333[298].fHigh := 39.841285;
    stLENS3_333[299].fEnergy := 17273.911917; stLENS3_333[299].fLow := 12.329275; stLENS3_333[299].fHigh := 39.629686;
    stLENS3_333[300].fEnergy := 17308.494311; stLENS3_333[300].fLow := 12.282257; stLENS3_333[300].fHigh := 39.419371;
    stLENS3_333[301].fEnergy := 17343.145940; stLENS3_333[301].fLow := 12.235371; stLENS3_333[301].fHigh := 39.210332;
    stLENS3_333[302].fEnergy := 17377.866941; stLENS3_333[302].fLow := 12.188617; stLENS3_333[302].fHigh := 39.002559;
    stLENS3_333[303].fEnergy := 17412.657454; stLENS3_333[303].fLow := 12.141996; stLENS3_333[303].fHigh := 38.796045;
    stLENS3_333[304].fEnergy := 17447.517618; stLENS3_333[304].fLow := 12.095505; stLENS3_333[304].fHigh := 38.590781;
    stLENS3_333[305].fEnergy := 17482.447571; stLENS3_333[305].fLow := 12.049144; stLENS3_333[305].fHigh := 38.386760;
    stLENS3_333[306].fEnergy := 17517.447455; stLENS3_333[306].fLow := 12.002913; stLENS3_333[306].fHigh := 38.183972;
    stLENS3_333[307].fEnergy := 17552.517408; stLENS3_333[307].fLow := 11.956810; stLENS3_333[307].fHigh := 37.982410;
    stLENS3_333[308].fEnergy := 17587.657571; stLENS3_333[308].fLow := 11.910835; stLENS3_333[308].fHigh := 37.782065;
    stLENS3_333[309].fEnergy := 17622.868085; stLENS3_333[309].fLow := 11.864987; stLENS3_333[309].fHigh := 37.582930;
    stLENS3_333[310].fEnergy := 17658.149090; stLENS3_333[310].fLow := 11.819266; stLENS3_333[310].fHigh := 37.384996;
    stLENS3_333[311].fEnergy := 17693.500728; stLENS3_333[311].fLow := 11.773670; stLENS3_333[311].fHigh := 37.188256;
    stLENS3_333[312].fEnergy := 17728.923140; stLENS3_333[312].fLow := 11.728199; stLENS3_333[312].fHigh := 36.992701;
    stLENS3_333[313].fEnergy := 17764.416468; stLENS3_333[313].fLow := 11.682853; stLENS3_333[313].fHigh := 36.798324;
    stLENS3_333[314].fEnergy := 17799.980854; stLENS3_333[314].fLow := 11.637630; stLENS3_333[314].fHigh := 36.605118;
    stLENS3_333[315].fEnergy := 17835.616439; stLENS3_333[315].fLow := 11.592530; stLENS3_333[315].fHigh := 36.413074;
    stLENS3_333[316].fEnergy := 17871.323367; stLENS3_333[316].fLow := 11.547553; stLENS3_333[316].fHigh := 36.222184;
    stLENS3_333[317].fEnergy := 17907.101780; stLENS3_333[317].fLow := 11.502697; stLENS3_333[317].fHigh := 36.032442;
    stLENS3_333[318].fEnergy := 17942.951822; stLENS3_333[318].fLow := 11.457962; stLENS3_333[318].fHigh := 35.843839;
    stLENS3_333[319].fEnergy := 17978.873635; stLENS3_333[319].fLow := 11.413347; stLENS3_333[319].fHigh := 35.656368;
    stLENS3_333[320].fEnergy := 18014.867364; stLENS3_333[320].fLow := 11.368852; stLENS3_333[320].fHigh := 35.470022;
    stLENS3_333[321].fEnergy := 18050.933153; stLENS3_333[321].fLow := 11.324477; stLENS3_333[321].fHigh := 35.284793;
    stLENS3_333[322].fEnergy := 18087.071145; stLENS3_333[322].fLow := 11.280219; stLENS3_333[322].fHigh := 35.100675;
    stLENS3_333[323].fEnergy := 18123.281486; stLENS3_333[323].fLow := 11.236080; stLENS3_333[323].fHigh := 34.917658;
    stLENS3_333[324].fEnergy := 18159.564319; stLENS3_333[324].fLow := 11.192057; stLENS3_333[324].fHigh := 34.735738;
    stLENS3_333[325].fEnergy := 18195.919791; stLENS3_333[325].fLow := 11.148151; stLENS3_333[325].fHigh := 34.554905;
    stLENS3_333[326].fEnergy := 18232.348047; stLENS3_333[326].fLow := 11.104362; stLENS3_333[326].fHigh := 34.375153;
    stLENS3_333[327].fEnergy := 18268.849232; stLENS3_333[327].fLow := 11.060687; stLENS3_333[327].fHigh := 34.196476;
    stLENS3_333[328].fEnergy := 18305.423493; stLENS3_333[328].fLow := 11.017128; stLENS3_333[328].fHigh := 34.018865;
    stLENS3_333[329].fEnergy := 18342.070975; stLENS3_333[329].fLow := 10.973683; stLENS3_333[329].fHigh := 33.842315;
    stLENS3_333[330].fEnergy := 18378.791826; stLENS3_333[330].fLow := 10.930351; stLENS3_333[330].fHigh := 33.666817;
    stLENS3_333[331].fEnergy := 18415.586191; stLENS3_333[331].fLow := 10.887133; stLENS3_333[331].fHigh := 33.492366;
    stLENS3_333[332].fEnergy := 18452.454219; stLENS3_333[332].fLow := 10.844027; stLENS3_333[332].fHigh := 33.318954;
    stLENS3_333[333].fEnergy := 18489.396057; stLENS3_333[333].fLow := 10.801034; stLENS3_333[333].fHigh := 33.146575;
    stLENS3_333[334].fEnergy := 18526.411853; stLENS3_333[334].fLow := 10.758151; stLENS3_333[334].fHigh := 32.975221;
    stLENS3_333[335].fEnergy := 18563.501754; stLENS3_333[335].fLow := 10.715380; stLENS3_333[335].fHigh := 32.804887;
    stLENS3_333[336].fEnergy := 18600.665909; stLENS3_333[336].fLow := 10.672720; stLENS3_333[336].fHigh := 32.635565;
    stLENS3_333[337].fEnergy := 18637.904467; stLENS3_333[337].fLow := 10.630169; stLENS3_333[337].fHigh := 32.467249;
    stLENS3_333[338].fEnergy := 18675.217577; stLENS3_333[338].fLow := 10.587728; stLENS3_333[338].fHigh := 32.299932;
    stLENS3_333[339].fEnergy := 18712.605388; stLENS3_333[339].fLow := 10.545396; stLENS3_333[339].fHigh := 32.133608;
    stLENS3_333[340].fEnergy := 18750.068048; stLENS3_333[340].fLow := 10.501307; stLENS3_333[340].fHigh := 31.968271;
    stLENS3_333[341].fEnergy := 18787.605710; stLENS3_333[341].fLow := 10.459865; stLENS3_333[341].fHigh := 31.803913;
    stLENS3_333[342].fEnergy := 18825.218521; stLENS3_333[342].fLow := 10.418586; stLENS3_333[342].fHigh := 31.640529;
    stLENS3_333[343].fEnergy := 18862.906634; stLENS3_333[343].fLow := 10.377471; stLENS3_333[343].fHigh := 31.478113;
    stLENS3_333[344].fEnergy := 18900.670198; stLENS3_333[344].fLow := 10.336517; stLENS3_333[344].fHigh := 31.316657;
    stLENS3_333[345].fEnergy := 18938.509365; stLENS3_333[345].fLow := 10.295725; stLENS3_333[345].fHigh := 31.156156;
    stLENS3_333[346].fEnergy := 18976.424286; stLENS3_333[346].fLow := 10.255094; stLENS3_333[346].fHigh := 30.996603;
    stLENS3_333[347].fEnergy := 19014.415113; stLENS3_333[347].fLow := 10.214624; stLENS3_333[347].fHigh := 30.837993;
    stLENS3_333[348].fEnergy := 19052.481997; stLENS3_333[348].fLow := 10.174313; stLENS3_333[348].fHigh := 30.680319;
    stLENS3_333[349].fEnergy := 19090.625092; stLENS3_333[349].fLow := 10.134161; stLENS3_333[349].fHigh := 30.523576;
    stLENS3_333[350].fEnergy := 19128.844549; stLENS3_333[350].fLow := 10.094168; stLENS3_333[350].fHigh := 30.367756;
    stLENS3_333[351].fEnergy := 19167.140521; stLENS3_333[351].fLow := 10.054332; stLENS3_333[351].fHigh := 30.212855;
    stLENS3_333[352].fEnergy := 19205.513162; stLENS3_333[352].fLow := 10.014654; stLENS3_333[352].fHigh := 30.058866;
    stLENS3_333[353].fEnergy := 19243.962625; stLENS3_333[353].fLow := 9.975132; stLENS3_333[353].fHigh := 29.905784;
    stLENS3_333[354].fEnergy := 19282.489064; stLENS3_333[354].fLow := 9.935767; stLENS3_333[354].fHigh := 29.753602;
    stLENS3_333[355].fEnergy := 19321.092632; stLENS3_333[355].fLow := 9.896556; stLENS3_333[355].fHigh := 29.602314;
    stLENS3_333[356].fEnergy := 19359.773486; stLENS3_333[356].fLow := 9.857501; stLENS3_333[356].fHigh := 29.451916;
    stLENS3_333[357].fEnergy := 19398.531778; stLENS3_333[357].fLow := 9.818599; stLENS3_333[357].fHigh := 29.302401;
    stLENS3_333[358].fEnergy := 19437.367665; stLENS3_333[358].fLow := 9.779851; stLENS3_333[358].fHigh := 29.153763;
    stLENS3_333[359].fEnergy := 19476.281301; stLENS3_333[359].fLow := 9.741256; stLENS3_333[359].fHigh := 29.005997;
    stLENS3_333[360].fEnergy := 19515.272842; stLENS3_333[360].fLow := 9.702813; stLENS3_333[360].fHigh := 28.859098;
    stLENS3_333[361].fEnergy := 19554.342444; stLENS3_333[361].fLow := 9.664522; stLENS3_333[361].fHigh := 28.713059;
    stLENS3_333[362].fEnergy := 19593.490264; stLENS3_333[362].fLow := 9.626382; stLENS3_333[362].fHigh := 28.567875;
    stLENS3_333[363].fEnergy := 19632.716457; stLENS3_333[363].fLow := 9.588393; stLENS3_333[363].fHigh := 28.423540;
    stLENS3_333[364].fEnergy := 19672.021182; stLENS3_333[364].fLow := 9.550554; stLENS3_333[364].fHigh := 28.280050;
    stLENS3_333[365].fEnergy := 19711.404594; stLENS3_333[365].fLow := 9.512863; stLENS3_333[365].fHigh := 28.137399;
    stLENS3_333[366].fEnergy := 19750.866853; stLENS3_333[366].fLow := 9.475322; stLENS3_333[366].fHigh := 27.995581;
    stLENS3_333[367].fEnergy := 19790.408115; stLENS3_333[367].fLow := 9.437929; stLENS3_333[367].fHigh := 27.854591;
    stLENS3_333[368].fEnergy := 19830.028538; stLENS3_333[368].fLow := 9.400683; stLENS3_333[368].fHigh := 27.714423;
    stLENS3_333[369].fEnergy := 19869.728282; stLENS3_333[369].fLow := 9.363584; stLENS3_333[369].fHigh := 27.575073;
    stLENS3_333[370].fEnergy := 19909.507504; stLENS3_333[370].fLow := 9.326632; stLENS3_333[370].fHigh := 27.436535;
    stLENS3_333[371].fEnergy := 19949.366365; stLENS3_333[371].fLow := 9.289825; stLENS3_333[371].fHigh := 27.298804;
    stLENS3_333[372].fEnergy := 19989.305023; stLENS3_333[372].fLow := 9.253164; stLENS3_333[372].fHigh := 27.161875;
    stLENS3_333[373].fEnergy := 20029.323638; stLENS3_333[373].fLow := 9.216648; stLENS3_333[373].fHigh := 27.025742;
    stLENS3_333[374].fEnergy := 20069.422371; stLENS3_333[374].fLow := 9.180275; stLENS3_333[374].fHigh := 26.890402;
    stLENS3_333[375].fEnergy := 20109.601381; stLENS3_333[375].fLow := 9.144046; stLENS3_333[375].fHigh := 26.755847;
    stLENS3_333[376].fEnergy := 20149.860830; stLENS3_333[376].fLow := 9.107960; stLENS3_333[376].fHigh := 26.622074;
    stLENS3_333[377].fEnergy := 20190.200878; stLENS3_333[377].fLow := 9.072017; stLENS3_333[377].fHigh := 26.489077;
    stLENS3_333[378].fEnergy := 20230.621687; stLENS3_333[378].fLow := 9.036215; stLENS3_333[378].fHigh := 26.356852;
    stLENS3_333[379].fEnergy := 20271.123419; stLENS3_333[379].fLow := 9.000555; stLENS3_333[379].fHigh := 26.225394;
    stLENS3_333[380].fEnergy := 20311.706235; stLENS3_333[380].fLow := 8.965035; stLENS3_333[380].fHigh := 26.094697;
    stLENS3_333[381].fEnergy := 20352.370298; stLENS3_333[381].fLow := 8.929656; stLENS3_333[381].fHigh := 25.964757;
    stLENS3_333[382].fEnergy := 20393.115770; stLENS3_333[382].fLow := 8.894416; stLENS3_333[382].fHigh := 25.835570;
    stLENS3_333[383].fEnergy := 20433.942815; stLENS3_333[383].fLow := 8.859315; stLENS3_333[383].fHigh := 25.707129;
    stLENS3_333[384].fEnergy := 20474.851596; stLENS3_333[384].fLow := 8.824353; stLENS3_333[384].fHigh := 25.579431;
    stLENS3_333[385].fEnergy := 20515.842276; stLENS3_333[385].fLow := 8.789528; stLENS3_333[385].fHigh := 25.452470;
    stLENS3_333[386].fEnergy := 20556.915020; stLENS3_333[386].fLow := 8.754842; stLENS3_333[386].fHigh := 25.326243;
    stLENS3_333[387].fEnergy := 20598.069991; stLENS3_333[387].fLow := 8.720292; stLENS3_333[387].fHigh := 25.200744;
    stLENS3_333[388].fEnergy := 20639.307355; stLENS3_333[388].fLow := 8.685878; stLENS3_333[388].fHigh := 25.075969;
    stLENS3_333[389].fEnergy := 20680.627276; stLENS3_333[389].fLow := 8.651600; stLENS3_333[389].fHigh := 24.951913;
    stLENS3_333[390].fEnergy := 20722.029919; stLENS3_333[390].fLow := 8.617458; stLENS3_333[390].fHigh := 24.828572;
    stLENS3_333[391].fEnergy := 20763.515451; stLENS3_333[391].fLow := 8.583450; stLENS3_333[391].fHigh := 24.705941;
    stLENS3_333[392].fEnergy := 20805.084036; stLENS3_333[392].fLow := 8.549576; stLENS3_333[392].fHigh := 24.584015;
    stLENS3_333[393].fEnergy := 20846.735842; stLENS3_333[393].fLow := 8.515836; stLENS3_333[393].fHigh := 24.462791;
    stLENS3_333[394].fEnergy := 20888.471035; stLENS3_333[394].fLow := 8.482229; stLENS3_333[394].fHigh := 24.342263;
    stLENS3_333[395].fEnergy := 20930.289782; stLENS3_333[395].fLow := 8.448755; stLENS3_333[395].fHigh := 24.222427;
    stLENS3_333[396].fEnergy := 20972.192250; stLENS3_333[396].fLow := 8.415413; stLENS3_333[396].fHigh := 24.103279;
    stLENS3_333[397].fEnergy := 21014.178607; stLENS3_333[397].fLow := 8.382203; stLENS3_333[397].fHigh := 23.984815;
    stLENS3_333[398].fEnergy := 21056.249021; stLENS3_333[398].fLow := 8.349123; stLENS3_333[398].fHigh := 23.867030;
    stLENS3_333[399].fEnergy := 21098.403659; stLENS3_333[399].fLow := 8.316175; stLENS3_333[399].fHigh := 23.749920;
    stLENS3_333[400].fEnergy := 21140.642692; stLENS3_333[400].fLow := 8.283356; stLENS3_333[400].fHigh := 23.633481;
    stLENS3_333[401].fEnergy := 21182.966286; stLENS3_333[401].fLow := 8.250666; stLENS3_333[401].fHigh := 23.517708;
    stLENS3_333[402].fEnergy := 21225.374613; stLENS3_333[402].fLow := 8.218106; stLENS3_333[402].fHigh := 23.402598;
    stLENS3_333[403].fEnergy := 21267.867841; stLENS3_333[403].fLow := 8.185674; stLENS3_333[403].fHigh := 23.288145;
    stLENS3_333[404].fEnergy := 21310.446141; stLENS3_333[404].fLow := 8.153370; stLENS3_333[404].fHigh := 23.174346;
    stLENS3_333[405].fEnergy := 21353.109683; stLENS3_333[405].fLow := 8.121194; stLENS3_333[405].fHigh := 23.061197;
    stLENS3_333[406].fEnergy := 21395.858637; stLENS3_333[406].fLow := 8.089145; stLENS3_333[406].fHigh := 22.948694;
    stLENS3_333[407].fEnergy := 21438.693174; stLENS3_333[407].fLow := 8.057222; stLENS3_333[407].fHigh := 22.836833;
    stLENS3_333[408].fEnergy := 21481.613467; stLENS3_333[408].fLow := 8.025425; stLENS3_333[408].fHigh := 22.725609;
    stLENS3_333[409].fEnergy := 21524.619686; stLENS3_333[409].fLow := 7.993754; stLENS3_333[409].fHigh := 22.615018;
    stLENS3_333[410].fEnergy := 21567.712003; stLENS3_333[410].fLow := 7.962207; stLENS3_333[410].fHigh := 22.505058;
    stLENS3_333[411].fEnergy := 21610.890591; stLENS3_333[411].fLow := 7.930785; stLENS3_333[411].fHigh := 22.395723;
    stLENS3_333[412].fEnergy := 21654.155623; stLENS3_333[412].fLow := 7.899487; stLENS3_333[412].fHigh := 22.287009;
    stLENS3_333[413].fEnergy := 21697.507271; stLENS3_333[413].fLow := 7.868313; stLENS3_333[413].fHigh := 22.178914;
    stLENS3_333[414].fEnergy := 21740.945710; stLENS3_333[414].fLow := 7.837261; stLENS3_333[414].fHigh := 22.071432;
    stLENS3_333[415].fEnergy := 21784.471112; stLENS3_333[415].fLow := 7.806333; stLENS3_333[415].fHigh := 21.964561;
    stLENS3_333[416].fEnergy := 21828.083652; stLENS3_333[416].fLow := 7.775526; stLENS3_333[416].fHigh := 21.858296;
    stLENS3_333[417].fEnergy := 21871.783505; stLENS3_333[417].fLow := 7.744841; stLENS3_333[417].fHigh := 21.752633;
    stLENS3_333[418].fEnergy := 21915.570845; stLENS3_333[418].fLow := 7.714276; stLENS3_333[418].fHigh := 21.647570;
    stLENS3_333[419].fEnergy := 21959.445847; stLENS3_333[419].fLow := 7.683833; stLENS3_333[419].fHigh := 21.543101;
    stLENS3_333[420].fEnergy := 22003.408687; stLENS3_333[420].fLow := 7.653510; stLENS3_333[420].fHigh := 21.439223;
    stLENS3_333[421].fEnergy := 22047.459540; stLENS3_333[421].fLow := 7.623306; stLENS3_333[421].fHigh := 21.335933;
    stLENS3_333[422].fEnergy := 22091.598584; stLENS3_333[422].fLow := 7.593221; stLENS3_333[422].fHigh := 21.233227;
    stLENS3_333[423].fEnergy := 22135.825994; stLENS3_333[423].fLow := 7.563256; stLENS3_333[423].fHigh := 21.131101;
    stLENS3_333[424].fEnergy := 22180.141947; stLENS3_333[424].fLow := 7.533408; stLENS3_333[424].fHigh := 21.029552;
    stLENS3_333[425].fEnergy := 22224.546620; stLENS3_333[425].fLow := 7.503678; stLENS3_333[425].fHigh := 20.928576;
    stLENS3_333[426].fEnergy := 22269.040192; stLENS3_333[426].fLow := 7.474066; stLENS3_333[426].fHigh := 20.828169;
    stLENS3_333[427].fEnergy := 22313.622841; stLENS3_333[427].fLow := 7.444570; stLENS3_333[427].fHigh := 20.728329;
    stLENS3_333[428].fEnergy := 22358.294743; stLENS3_333[428].fLow := 7.415191; stLENS3_333[428].fHigh := 20.629051;
    stLENS3_333[429].fEnergy := 22403.056079; stLENS3_333[429].fLow := 7.385928; stLENS3_333[429].fHigh := 20.530331;
    stLENS3_333[430].fEnergy := 22447.907027; stLENS3_333[430].fLow := 7.356780; stLENS3_333[430].fHigh := 20.432167;
    stLENS3_333[431].fEnergy := 22492.847767; stLENS3_333[431].fLow := 7.327748; stLENS3_333[431].fHigh := 20.334556;
    stLENS3_333[432].fEnergy := 22537.878478; stLENS3_333[432].fLow := 7.298829; stLENS3_333[432].fHigh := 20.237492;
    stLENS3_333[433].fEnergy := 22582.999341; stLENS3_333[433].fLow := 7.270025; stLENS3_333[433].fHigh := 20.140974;
    stLENS3_333[434].fEnergy := 22628.210536; stLENS3_333[434].fLow := 7.241335; stLENS3_333[434].fHigh := 20.044998;
    stLENS3_333[435].fEnergy := 22673.512244; stLENS3_333[435].fLow := 7.212758; stLENS3_333[435].fHigh := 19.949560;
    stLENS3_333[436].fEnergy := 22718.904645; stLENS3_333[436].fLow := 7.184294; stLENS3_333[436].fHigh := 19.854657;
    stLENS3_333[437].fEnergy := 22764.387923; stLENS3_333[437].fLow := 7.155942; stLENS3_333[437].fHigh := 19.760286;
    stLENS3_333[438].fEnergy := 22809.962258; stLENS3_333[438].fLow := 7.127702; stLENS3_333[438].fHigh := 19.666443;
    stLENS3_333[439].fEnergy := 22855.627833; stLENS3_333[439].fLow := 7.099573; stLENS3_333[439].fHigh := 19.573126;
    stLENS3_333[440].fEnergy := 22901.384830; stLENS3_333[440].fLow := 7.071555; stLENS3_333[440].fHigh := 19.480330;
    stLENS3_333[441].fEnergy := 22947.233433; stLENS3_333[441].fLow := 7.043648; stLENS3_333[441].fHigh := 19.388053;
    stLENS3_333[442].fEnergy := 22993.173825; stLENS3_333[442].fLow := 7.015851; stLENS3_333[442].fHigh := 19.296292;
    stLENS3_333[443].fEnergy := 23039.206190; stLENS3_333[443].fLow := 6.988164; stLENS3_333[443].fHigh := 19.205043;
    stLENS3_333[444].fEnergy := 23085.330711; stLENS3_333[444].fLow := 6.960586; stLENS3_333[444].fHigh := 19.114303;
    stLENS3_333[445].fEnergy := 23131.547574; stLENS3_333[445].fLow := 6.933117; stLENS3_333[445].fHigh := 19.024070;
    stLENS3_333[446].fEnergy := 23177.856963; stLENS3_333[446].fLow := 6.905756; stLENS3_333[446].fHigh := 18.934339;
    stLENS3_333[447].fEnergy := 23224.259064; stLENS3_333[447].fLow := 6.878503; stLENS3_333[447].fHigh := 18.845108;
    stLENS3_333[448].fEnergy := 23270.754061; stLENS3_333[448].fLow := 6.851358; stLENS3_333[448].fHigh := 18.756374;
    stLENS3_333[449].fEnergy := 23317.342142; stLENS3_333[449].fLow := 6.824320; stLENS3_333[449].fHigh := 18.668133;
    stLENS3_333[450].fEnergy := 23364.023492; stLENS3_333[450].fLow := 6.797389; stLENS3_333[450].fHigh := 18.580383;
    stLENS3_333[451].fEnergy := 23410.798298; stLENS3_333[451].fLow := 6.770564; stLENS3_333[451].fHigh := 18.493121;
    stLENS3_333[452].fEnergy := 23457.666748; stLENS3_333[452].fLow := 6.743844; stLENS3_333[452].fHigh := 18.406343;
    stLENS3_333[453].fEnergy := 23504.629028; stLENS3_333[453].fLow := 6.717230; stLENS3_333[453].fHigh := 18.320047;
    stLENS3_333[454].fEnergy := 23551.685327; stLENS3_333[454].fLow := 6.690722; stLENS3_333[454].fHigh := 18.234229;
    stLENS3_333[455].fEnergy := 23598.835832; stLENS3_333[455].fLow := 6.664318; stLENS3_333[455].fHigh := 18.148888;
    stLENS3_333[456].fEnergy := 23646.080733; stLENS3_333[456].fLow := 6.638018; stLENS3_333[456].fHigh := 18.064019;
    stLENS3_333[457].fEnergy := 23693.420218; stLENS3_333[457].fLow := 6.611821; stLENS3_333[457].fHigh := 17.979620;
    stLENS3_333[458].fEnergy := 23740.854477; stLENS3_333[458].fLow := 6.585729; stLENS3_333[458].fHigh := 17.895688;
    stLENS3_333[459].fEnergy := 23788.383699; stLENS3_333[459].fLow := 6.559739; stLENS3_333[459].fHigh := 17.812221;
    stLENS3_333[460].fEnergy := 23836.008075; stLENS3_333[460].fLow := 6.533851; stLENS3_333[460].fHigh := 17.729214;
    stLENS3_333[461].fEnergy := 23883.727795; stLENS3_333[461].fLow := 6.508066; stLENS3_333[461].fHigh := 17.646667;
    stLENS3_333[462].fEnergy := 23931.543050; stLENS3_333[462].fLow := 6.482383; stLENS3_333[462].fHigh := 17.564575;
    stLENS3_333[463].fEnergy := 23979.454031; stLENS3_333[463].fLow := 6.456801; stLENS3_333[463].fHigh := 17.482935;
    stLENS3_333[464].fEnergy := 24027.460930; stLENS3_333[464].fLow := 6.431320; stLENS3_333[464].fHigh := 17.401746;
    stLENS3_333[465].fEnergy := 24075.563939; stLENS3_333[465].fLow := 6.405940; stLENS3_333[465].fHigh := 17.321005;
    stLENS3_333[466].fEnergy := 24123.763250; stLENS3_333[466].fLow := 6.380659; stLENS3_333[466].fHigh := 17.240708;
    stLENS3_333[467].fEnergy := 24172.059056; stLENS3_333[467].fLow := 6.355479; stLENS3_333[467].fHigh := 17.160853;
    stLENS3_333[468].fEnergy := 24220.451551; stLENS3_333[468].fLow := 6.330398; stLENS3_333[468].fHigh := 17.081438;
    stLENS3_333[469].fEnergy := 24268.940927; stLENS3_333[469].fLow := 6.305415; stLENS3_333[469].fHigh := 17.002459;
    stLENS3_333[470].fEnergy := 24317.527379; stLENS3_333[470].fLow := 6.280532; stLENS3_333[470].fHigh := 16.923914;
    stLENS3_333[471].fEnergy := 24366.211101; stLENS3_333[471].fLow := 6.255746; stLENS3_333[471].fHigh := 16.845800;
    stLENS3_333[472].fEnergy := 24414.992288; stLENS3_333[472].fLow := 6.231059; stLENS3_333[472].fHigh := 16.768115;
    stLENS3_333[473].fEnergy := 24463.871136; stLENS3_333[473].fLow := 6.206469; stLENS3_333[473].fHigh := 16.690856;
    stLENS3_333[474].fEnergy := 24512.847838; stLENS3_333[474].fLow := 6.181976; stLENS3_333[474].fHigh := 16.614020;
    stLENS3_333[475].fEnergy := 24561.922592; stLENS3_333[475].fLow := 6.157579; stLENS3_333[475].fHigh := 16.537606;
    stLENS3_333[476].fEnergy := 24611.095594; stLENS3_333[476].fLow := 6.133279; stLENS3_333[476].fHigh := 16.461610;
    stLENS3_333[477].fEnergy := 24660.367040; stLENS3_333[477].fLow := 6.109075; stLENS3_333[477].fHigh := 16.386029;
    stLENS3_333[478].fEnergy := 24709.737128; stLENS3_333[478].fLow := 6.084966; stLENS3_333[478].fHigh := 16.310862;
    stLENS3_333[479].fEnergy := 24759.206055; stLENS3_333[479].fLow := 6.060952; stLENS3_333[479].fHigh := 16.236106;
    stLENS3_333[480].fEnergy := 24808.774018; stLENS3_333[480].fLow := 6.037033; stLENS3_333[480].fHigh := 16.161758;
    stLENS3_333[481].fEnergy := 24858.441217; stLENS3_333[481].fLow := 6.013209; stLENS3_333[481].fHigh := 16.087815;
    stLENS3_333[482].fEnergy := 24908.207849; stLENS3_333[482].fLow := 5.989478; stLENS3_333[482].fHigh := 16.014277;
    stLENS3_333[483].fEnergy := 24958.074115; stLENS3_333[483].fLow := 5.965842; stLENS3_333[483].fHigh := 15.941139;
    stLENS3_333[484].fEnergy := 25008.040212; stLENS3_333[484].fLow := 5.942298; stLENS3_333[484].fHigh := 15.868399;
    stLENS3_333[485].fEnergy := 25058.106342; stLENS3_333[485].fLow := 5.918848; stLENS3_333[485].fHigh := 15.796056;
    stLENS3_333[486].fEnergy := 25108.272705; stLENS3_333[486].fLow := 5.895489; stLENS3_333[486].fHigh := 15.724106;
    stLENS3_333[487].fEnergy := 25158.539500; stLENS3_333[487].fLow := 5.872224; stLENS3_333[487].fHigh := 15.652548;
    stLENS3_333[488].fEnergy := 25208.906930; stLENS3_333[488].fLow := 5.849050; stLENS3_333[488].fHigh := 15.581379;
    stLENS3_333[489].fEnergy := 25259.375195; stLENS3_333[489].fLow := 5.825967; stLENS3_333[489].fHigh := 15.510596;
    stLENS3_333[490].fEnergy := 25309.944498; stLENS3_333[490].fLow := 5.802975; stLENS3_333[490].fHigh := 15.440198;
    stLENS3_333[491].fEnergy := 25360.615041; stLENS3_333[491].fLow := 5.780075; stLENS3_333[491].fHigh := 15.370181;
    stLENS3_333[492].fEnergy := 25411.387026; stLENS3_333[492].fLow := 5.757264; stLENS3_333[492].fHigh := 15.300545;
    stLENS3_333[493].fEnergy := 25462.260656; stLENS3_333[493].fLow := 5.734544; stLENS3_333[493].fHigh := 15.231285;
    stLENS3_333[494].fEnergy := 25513.236136; stLENS3_333[494].fLow := 5.711913; stLENS3_333[494].fHigh := 15.162401;
    stLENS3_333[495].fEnergy := 25564.313669; stLENS3_333[495].fLow := 5.689372; stLENS3_333[495].fHigh := 15.093890;
    stLENS3_333[496].fEnergy := 25615.493459; stLENS3_333[496].fLow := 5.666919; stLENS3_333[496].fHigh := 15.025749;
    stLENS3_333[497].fEnergy := 25666.775711; stLENS3_333[497].fLow := 5.644555; stLENS3_333[497].fHigh := 14.957977;
    stLENS3_333[498].fEnergy := 25718.160630; stLENS3_333[498].fLow := 5.622280; stLENS3_333[498].fHigh := 14.890570;
    stLENS3_333[499].fEnergy := 25769.648422; stLENS3_333[499].fLow := 5.600092; stLENS3_333[499].fHigh := 14.823528;
    stLENS3_333[500].fEnergy := 25821.239293; stLENS3_333[500].fLow := 5.577992; stLENS3_333[500].fHigh := 14.756848;
    stLENS3_333[501].fEnergy := 25872.933448; stLENS3_333[501].fLow := 5.555979; stLENS3_333[501].fHigh := 14.690527;
    stLENS3_333[502].fEnergy := 25924.731096; stLENS3_333[502].fLow := 5.534053; stLENS3_333[502].fHigh := 14.624564;
    stLENS3_333[503].fEnergy := 25976.632442; stLENS3_333[503].fLow := 5.512214; stLENS3_333[503].fHigh := 14.558956;
    stLENS3_333[504].fEnergy := 26028.637695; stLENS3_333[504].fLow := 5.490460; stLENS3_333[504].fHigh := 14.493702;
    stLENS3_333[505].fEnergy := 26080.747062; stLENS3_333[505].fLow := 5.468793; stLENS3_333[505].fHigh := 14.428798;
    stLENS3_333[506].fEnergy := 26132.960752; stLENS3_333[506].fLow := 5.447211; stLENS3_333[506].fHigh := 14.364244;
    stLENS3_333[507].fEnergy := 26185.278975; stLENS3_333[507].fLow := 5.425714; stLENS3_333[507].fHigh := 14.300036;
    stLENS3_333[508].fEnergy := 26237.701938; stLENS3_333[508].fLow := 5.404302; stLENS3_333[508].fHigh := 14.236173;
    stLENS3_333[509].fEnergy := 26290.229852; stLENS3_333[509].fLow := 5.382975; stLENS3_333[509].fHigh := 14.172653;
    stLENS3_333[510].fEnergy := 26342.862928; stLENS3_333[510].fLow := 5.361731; stLENS3_333[510].fHigh := 14.109474;
    stLENS3_333[511].fEnergy := 26395.601374; stLENS3_333[511].fLow := 5.340572; stLENS3_333[511].fHigh := 14.046634;
    stLENS3_333[512].fEnergy := 26448.445404; stLENS3_333[512].fLow := 5.319496; stLENS3_333[512].fHigh := 13.984130;
    stLENS3_333[513].fEnergy := 26501.395226; stLENS3_333[513].fLow := 5.298503; stLENS3_333[513].fHigh := 13.921961;
    stLENS3_333[514].fEnergy := 26554.451055; stLENS3_333[514].fLow := 5.277593; stLENS3_333[514].fHigh := 13.860124;
    stLENS3_333[515].fEnergy := 26607.613102; stLENS3_333[515].fLow := 5.256766; stLENS3_333[515].fHigh := 13.798619;
    stLENS3_333[516].fEnergy := 26660.881578; stLENS3_333[516].fLow := 5.236021; stLENS3_333[516].fHigh := 13.737442;
    stLENS3_333[517].fEnergy := 26714.256699; stLENS3_333[517].fLow := 5.215357; stLENS3_333[517].fHigh := 13.676592;
    stLENS3_333[518].fEnergy := 26767.738676; stLENS3_333[518].fLow := 5.194775; stLENS3_333[518].fHigh := 13.616067;
    stLENS3_333[519].fEnergy := 26821.327725; stLENS3_333[519].fLow := 5.174275; stLENS3_333[519].fHigh := 13.555865;
    stLENS3_333[520].fEnergy := 26875.024059; stLENS3_333[520].fLow := 5.153855; stLENS3_333[520].fHigh := 13.495983;
    stLENS3_333[521].fEnergy := 26928.827893; stLENS3_333[521].fLow := 5.133516; stLENS3_333[521].fHigh := 13.436421;
    stLENS3_333[522].fEnergy := 26982.739442; stLENS3_333[522].fLow := 5.113257; stLENS3_333[522].fHigh := 13.377176;
    stLENS3_333[523].fEnergy := 27036.758923; stLENS3_333[523].fLow := 5.093078; stLENS3_333[523].fHigh := 13.318247;
    stLENS3_333[524].fEnergy := 27090.886550; stLENS3_333[524].fLow := 5.072979; stLENS3_333[524].fHigh := 13.259631;
    stLENS3_333[525].fEnergy := 27145.122541; stLENS3_333[525].fLow := 5.052959; stLENS3_333[525].fHigh := 13.201326;
    stLENS3_333[526].fEnergy := 27199.467113; stLENS3_333[526].fLow := 5.033018; stLENS3_333[526].fHigh := 13.143332;
    stLENS3_333[527].fEnergy := 27253.920482; stLENS3_333[527].fLow := 5.013156; stLENS3_333[527].fHigh := 13.085645;
    stLENS3_333[528].fEnergy := 27308.482867; stLENS3_333[528].fLow := 4.993372; stLENS3_333[528].fHigh := 13.028264;
    stLENS3_333[529].fEnergy := 27363.154486; stLENS3_333[529].fLow := 4.973666; stLENS3_333[529].fHigh := 12.971188;
    stLENS3_333[530].fEnergy := 27417.935558; stLENS3_333[530].fLow := 4.954038; stLENS3_333[530].fHigh := 12.914414;
    stLENS3_333[531].fEnergy := 27472.826302; stLENS3_333[531].fLow := 4.934488; stLENS3_333[531].fHigh := 12.857941;
    stLENS3_333[532].fEnergy := 27527.826937; stLENS3_333[532].fLow := 4.915014; stLENS3_333[532].fHigh := 12.801767;
    stLENS3_333[533].fEnergy := 27582.937683; stLENS3_333[533].fLow := 4.895618; stLENS3_333[533].fHigh := 12.745890;
    stLENS3_333[534].fEnergy := 27638.158761; stLENS3_333[534].fLow := 4.876298; stLENS3_333[534].fHigh := 12.690309;
    stLENS3_333[535].fEnergy := 27693.490392; stLENS3_333[535].fLow := 4.857054; stLENS3_333[535].fHigh := 12.635022;
    stLENS3_333[536].fEnergy := 27748.932796; stLENS3_333[536].fLow := 4.837886; stLENS3_333[536].fHigh := 12.580026;
    stLENS3_333[537].fEnergy := 27804.486197; stLENS3_333[537].fLow := 4.818794; stLENS3_333[537].fHigh := 12.525321;
    stLENS3_333[538].fEnergy := 27860.150815; stLENS3_333[538].fLow := 4.799777; stLENS3_333[538].fHigh := 12.470904;
    stLENS3_333[539].fEnergy := 27915.926874; stLENS3_333[539].fLow := 4.780836; stLENS3_333[539].fHigh := 12.416774;
    stLENS3_333[540].fEnergy := 27971.814597; stLENS3_333[540].fLow := 4.761969; stLENS3_333[540].fHigh := 12.362929;
    stLENS3_333[541].fEnergy := 28027.814207; stLENS3_333[541].fLow := 4.743176; stLENS3_333[541].fHigh := 12.309368;
    stLENS3_333[542].fEnergy := 28083.925929; stLENS3_333[542].fLow := 4.724458; stLENS3_333[542].fHigh := 12.256088;
    stLENS3_333[543].fEnergy := 28140.149986; stLENS3_333[543].fLow := 4.705813; stLENS3_333[543].fHigh := 12.203089;
    stLENS3_333[544].fEnergy := 28196.486604; stLENS3_333[544].fLow := 4.687242; stLENS3_333[544].fHigh := 12.150369;
    stLENS3_333[545].fEnergy := 28252.936008; stLENS3_333[545].fLow := 4.668744; stLENS3_333[545].fHigh := 12.097925;
    stLENS3_333[546].fEnergy := 28309.498423; stLENS3_333[546].fLow := 4.650320; stLENS3_333[546].fHigh := 12.045757;
    stLENS3_333[547].fEnergy := 28366.174077; stLENS3_333[547].fLow := 4.631968; stLENS3_333[547].fHigh := 11.993862;
    stLENS3_333[548].fEnergy := 28422.963195; stLENS3_333[548].fLow := 4.613688; stLENS3_333[548].fHigh := 11.942239;
    stLENS3_333[549].fEnergy := 28479.866005; stLENS3_333[549].fLow := 4.595481; stLENS3_333[549].fHigh := 11.890887;
    stLENS3_333[550].fEnergy := 28536.882735; stLENS3_333[550].fLow := 4.577345; stLENS3_333[550].fHigh := 11.839804;
    stLENS3_333[551].fEnergy := 28594.013612; stLENS3_333[551].fLow := 4.559281; stLENS3_333[551].fHigh := 11.788988;
    stLENS3_333[552].fEnergy := 28651.258866; stLENS3_333[552].fLow := 4.541289; stLENS3_333[552].fHigh := 11.738438;
    stLENS3_333[553].fEnergy := 28708.618724; stLENS3_333[553].fLow := 4.523367; stLENS3_333[553].fHigh := 11.688153;
    stLENS3_333[554].fEnergy := 28766.093417; stLENS3_333[554].fLow := 4.505516; stLENS3_333[554].fHigh := 11.638130;
    stLENS3_333[555].fEnergy := 28823.683175; stLENS3_333[555].fLow := 4.487736; stLENS3_333[555].fHigh := 11.588368;
    stLENS3_333[556].fEnergy := 28881.388227; stLENS3_333[556].fLow := 4.470025; stLENS3_333[556].fHigh := 11.538866;
    stLENS3_333[557].fEnergy := 28939.208804; stLENS3_333[557].fLow := 4.452385; stLENS3_333[557].fHigh := 11.489621;
    stLENS3_333[558].fEnergy := 28997.145139; stLENS3_333[558].fLow := 4.434814; stLENS3_333[558].fHigh := 11.440634;
    stLENS3_333[559].fEnergy := 29055.197462; stLENS3_333[559].fLow := 4.417312; stLENS3_333[559].fHigh := 11.391902;
    stLENS3_333[560].fEnergy := 29113.366006; stLENS3_333[560].fLow := 4.399880; stLENS3_333[560].fHigh := 11.343423;
    stLENS3_333[561].fEnergy := 29171.651004; stLENS3_333[561].fLow := 4.382516; stLENS3_333[561].fHigh := 11.295197;
    stLENS3_333[562].fEnergy := 29230.052688; stLENS3_333[562].fLow := 4.365221; stLENS3_333[562].fHigh := 11.247221;
    stLENS3_333[563].fEnergy := 29288.571293; stLENS3_333[563].fLow := 4.347994; stLENS3_333[563].fHigh := 11.199495;
    stLENS3_333[564].fEnergy := 29347.207052; stLENS3_333[564].fLow := 4.330836; stLENS3_333[564].fHigh := 11.152016;
    stLENS3_333[565].fEnergy := 29405.960199; stLENS3_333[565].fLow := 4.313744; stLENS3_333[565].fHigh := 11.104784;
    stLENS3_333[566].fEnergy := 29464.830971; stLENS3_333[566].fLow := 4.296721; stLENS3_333[566].fHigh := 11.057797;
    stLENS3_333[567].fEnergy := 29523.819602; stLENS3_333[567].fLow := 4.279764; stLENS3_333[567].fHigh := 11.011054;
    stLENS3_333[568].fEnergy := 29582.926328; stLENS3_333[568].fLow := 4.262875; stLENS3_333[568].fHigh := 10.964552;
    stLENS3_333[569].fEnergy := 29642.151386; stLENS3_333[569].fLow := 4.246052; stLENS3_333[569].fHigh := 10.918292;
    stLENS3_333[570].fEnergy := 29701.495012; stLENS3_333[570].fLow := 4.229295; stLENS3_333[570].fHigh := 10.872270;
    stLENS3_333[571].fEnergy := 29760.957445; stLENS3_333[571].fLow := 4.212605; stLENS3_333[571].fHigh := 10.826487;
    stLENS3_333[572].fEnergy := 29820.538922; stLENS3_333[572].fLow := 4.195980; stLENS3_333[572].fHigh := 10.780940;
    stLENS3_333[573].fEnergy := 29880.239680; stLENS3_333[573].fLow := 4.179421; stLENS3_333[573].fHigh := 10.735629;
    stLENS3_333[574].fEnergy := 29940.059960; stLENS3_333[574].fLow := 4.162928; stLENS3_333[574].fHigh := 10.690551;
    stLENS3_333[575].fEnergy := 30000.000000; stLENS3_333[575].fLow := 4.146499; stLENS3_333[575].fHigh := 10.645706;
    stLENS3_333[576].fEnergy := 30068.760232; stLENS3_333[576].fLow := 4.127773; stLENS3_333[576].fHigh := 10.593372;
    stLENS3_333[577].fEnergy := 30128.957930; stLENS3_333[577].fLow := 4.111483; stLENS3_333[577].fHigh := 10.548614;
    stLENS3_333[578].fEnergy := 30189.276144; stLENS3_333[578].fLow := 4.095258; stLENS3_333[578].fHigh := 10.504044;
    stLENS3_333[579].fEnergy := 30249.715115; stLENS3_333[579].fLow := 4.079096; stLENS3_333[579].fHigh := 10.459662;
    stLENS3_333[580].fEnergy := 30310.275085; stLENS3_333[580].fLow := 4.062999; stLENS3_333[580].fHigh := 10.415468;
    stLENS3_333[581].fEnergy := 30370.956297; stLENS3_333[581].fLow := 4.046964; stLENS3_333[581].fHigh := 10.371461;
    stLENS3_333[582].fEnergy := 30431.758992; stLENS3_333[582].fLow := 4.030994; stLENS3_333[582].fHigh := 10.327640;
    stLENS3_333[583].fEnergy := 30492.683414; stLENS3_333[583].fLow := 4.015086; stLENS3_333[583].fHigh := 10.284004;
    stLENS3_333[584].fEnergy := 30553.729807; stLENS3_333[584].fLow := 3.999241; stLENS3_333[584].fHigh := 10.240552;
    stLENS3_333[585].fEnergy := 30614.898414; stLENS3_333[585].fLow := 3.983458; stLENS3_333[585].fHigh := 10.197284;
    stLENS3_333[586].fEnergy := 30676.189482; stLENS3_333[586].fLow := 3.967738; stLENS3_333[586].fHigh := 10.154198;
    stLENS3_333[587].fEnergy := 30737.603254; stLENS3_333[587].fLow := 3.952080; stLENS3_333[587].fHigh := 10.111295;
    stLENS3_333[588].fEnergy := 30799.139977; stLENS3_333[588].fLow := 3.936483; stLENS3_333[588].fHigh := 10.068573;
    stLENS3_333[589].fEnergy := 30860.799896; stLENS3_333[589].fLow := 3.920948; stLENS3_333[589].fHigh := 10.026031;
    stLENS3_333[590].fEnergy := 30922.583259; stLENS3_333[590].fLow := 3.905475; stLENS3_333[590].fHigh := 9.983669;
    stLENS3_333[591].fEnergy := 30984.490312; stLENS3_333[591].fLow := 3.890062; stLENS3_333[591].fHigh := 9.941487;
    stLENS3_333[592].fEnergy := 31046.521303; stLENS3_333[592].fLow := 3.874711; stLENS3_333[592].fHigh := 9.899482;
    stLENS3_333[593].fEnergy := 31108.676480; stLENS3_333[593].fLow := 3.859419; stLENS3_333[593].fHigh := 9.857655;
    stLENS3_333[594].fEnergy := 31170.956091; stLENS3_333[594].fLow := 3.844189; stLENS3_333[594].fHigh := 9.816005;
    stLENS3_333[595].fEnergy := 31233.360387; stLENS3_333[595].fLow := 3.829018; stLENS3_333[595].fHigh := 9.774530;
    stLENS3_333[596].fEnergy := 31295.889616; stLENS3_333[596].fLow := 3.813907; stLENS3_333[596].fHigh := 9.733231;
    stLENS3_333[597].fEnergy := 31358.544029; stLENS3_333[597].fLow := 3.798856; stLENS3_333[597].fHigh := 9.692106;
    stLENS3_333[598].fEnergy := 31421.323876; stLENS3_333[598].fLow := 3.783864; stLENS3_333[598].fHigh := 9.651155;
    stLENS3_333[599].fEnergy := 31484.229408; stLENS3_333[599].fLow := 3.768932; stLENS3_333[599].fHigh := 9.610378;
    stLENS3_333[600].fEnergy := 31547.260878; stLENS3_333[600].fLow := 3.754058; stLENS3_333[600].fHigh := 9.569772;
    stLENS3_333[601].fEnergy := 31610.418536; stLENS3_333[601].fLow := 3.739243; stLENS3_333[601].fHigh := 9.529338;
    stLENS3_333[602].fEnergy := 31673.702636; stLENS3_333[602].fLow := 3.724487; stLENS3_333[602].fHigh := 9.489075;
    stLENS3_333[603].fEnergy := 31737.113431; stLENS3_333[603].fLow := 3.709788; stLENS3_333[603].fHigh := 9.448982;
    stLENS3_333[604].fEnergy := 31800.651174; stLENS3_333[604].fLow := 3.695148; stLENS3_333[604].fHigh := 9.409058;
    stLENS3_333[605].fEnergy := 31864.316120; stLENS3_333[605].fLow := 3.680566; stLENS3_333[605].fHigh := 9.369303;
    stLENS3_333[606].fEnergy := 31928.108524; stLENS3_333[606].fLow := 3.666041; stLENS3_333[606].fHigh := 9.329716;
    stLENS3_333[607].fEnergy := 31992.028640; stLENS3_333[607].fLow := 3.651573; stLENS3_333[607].fHigh := 9.290296;
    stLENS3_333[608].fEnergy := 32056.076724; stLENS3_333[608].fLow := 3.637163; stLENS3_333[608].fHigh := 9.251043;
    stLENS3_333[609].fEnergy := 32120.253032; stLENS3_333[609].fLow := 3.622809; stLENS3_333[609].fHigh := 9.211956;
    stLENS3_333[610].fEnergy := 32184.557822; stLENS3_333[610].fLow := 3.608512; stLENS3_333[610].fHigh := 9.173034;
    stLENS3_333[611].fEnergy := 32248.991349; stLENS3_333[611].fLow := 3.594271; stLENS3_333[611].fHigh := 9.134276;
    stLENS3_333[612].fEnergy := 32313.553873; stLENS3_333[612].fLow := 3.580087; stLENS3_333[612].fHigh := 9.095682;
    stLENS3_333[613].fEnergy := 32378.245651; stLENS3_333[613].fLow := 3.565959; stLENS3_333[613].fHigh := 9.057251;
    stLENS3_333[614].fEnergy := 32443.066942; stLENS3_333[614].fLow := 3.551886; stLENS3_333[614].fHigh := 9.018982;
    stLENS3_333[615].fEnergy := 32508.018005; stLENS3_333[615].fLow := 3.537869; stLENS3_333[615].fHigh := 8.980876;
    stLENS3_333[616].fEnergy := 32573.099101; stLENS3_333[616].fLow := 3.523907; stLENS3_333[616].fHigh := 8.942930;
    stLENS3_333[617].fEnergy := 32638.310488; stLENS3_333[617].fLow := 3.510000; stLENS3_333[617].fHigh := 8.905144;
    stLENS3_333[618].fEnergy := 32703.652430; stLENS3_333[618].fLow := 3.496149; stLENS3_333[618].fHigh := 8.867518;
    stLENS3_333[619].fEnergy := 32769.125185; stLENS3_333[619].fLow := 3.482351; stLENS3_333[619].fHigh := 8.830052;
    stLENS3_333[620].fEnergy := 32834.729018; stLENS3_333[620].fLow := 3.468609; stLENS3_333[620].fHigh := 8.792743;
    stLENS3_333[621].fEnergy := 32900.464189; stLENS3_333[621].fLow := 3.454920; stLENS3_333[621].fHigh := 8.755592;
    stLENS3_333[622].fEnergy := 32966.330962; stLENS3_333[622].fLow := 3.441286; stLENS3_333[622].fHigh := 8.718598;
    stLENS3_333[623].fEnergy := 33032.329601; stLENS3_333[623].fLow := 3.427705; stLENS3_333[623].fHigh := 8.681760;
    stLENS3_333[624].fEnergy := 33098.460369; stLENS3_333[624].fLow := 3.414178; stLENS3_333[624].fHigh := 8.645078;
    stLENS3_333[625].fEnergy := 33164.723530; stLENS3_333[625].fLow := 3.400704; stLENS3_333[625].fHigh := 8.608551;
    stLENS3_333[626].fEnergy := 33231.119351; stLENS3_333[626].fLow := 3.387284; stLENS3_333[626].fHigh := 8.572179;
    stLENS3_333[627].fEnergy := 33297.648096; stLENS3_333[627].fLow := 3.373916; stLENS3_333[627].fHigh := 8.535960;
    stLENS3_333[628].fEnergy := 33364.310032; stLENS3_333[628].fLow := 3.360602; stLENS3_333[628].fHigh := 8.499894;
    stLENS3_333[629].fEnergy := 33431.105426; stLENS3_333[629].fLow := 3.347339; stLENS3_333[629].fHigh := 8.463980;
    stLENS3_333[630].fEnergy := 33498.034543; stLENS3_333[630].fLow := 3.334129; stLENS3_333[630].fHigh := 8.428218;
    stLENS3_333[631].fEnergy := 33565.097653; stLENS3_333[631].fLow := 3.320972; stLENS3_333[631].fHigh := 8.392608;
    stLENS3_333[632].fEnergy := 33632.295023; stLENS3_333[632].fLow := 3.307866; stLENS3_333[632].fHigh := 8.357147;
    stLENS3_333[633].fEnergy := 33699.626923; stLENS3_333[633].fLow := 3.294812; stLENS3_333[633].fHigh := 8.321837;
    stLENS3_333[634].fEnergy := 33767.093621; stLENS3_333[634].fLow := 3.281809; stLENS3_333[634].fHigh := 8.286676;
    stLENS3_333[635].fEnergy := 33834.695387; stLENS3_333[635].fLow := 3.268858; stLENS3_333[635].fHigh := 8.251663;
    stLENS3_333[636].fEnergy := 33902.432493; stLENS3_333[636].fLow := 3.255958; stLENS3_333[636].fHigh := 8.216798;
    stLENS3_333[637].fEnergy := 33970.305208; stLENS3_333[637].fLow := 3.243108; stLENS3_333[637].fHigh := 8.182081;
    stLENS3_333[638].fEnergy := 34038.313804; stLENS3_333[638].fLow := 3.230310; stLENS3_333[638].fHigh := 8.147510;
    stLENS3_333[639].fEnergy := 34106.458554; stLENS3_333[639].fLow := 3.217562; stLENS3_333[639].fHigh := 8.113085;
    stLENS3_333[640].fEnergy := 34174.739729; stLENS3_333[640].fLow := 3.204864; stLENS3_333[640].fHigh := 8.078806;
    stLENS3_333[641].fEnergy := 34243.157604; stLENS3_333[641].fLow := 3.192216; stLENS3_333[641].fHigh := 8.044671;
    stLENS3_333[642].fEnergy := 34311.712451; stLENS3_333[642].fLow := 3.179619; stLENS3_333[642].fHigh := 8.010681;
    stLENS3_333[643].fEnergy := 34380.404545; stLENS3_333[643].fLow := 3.167071; stLENS3_333[643].fHigh := 7.976835;
    stLENS3_333[644].fEnergy := 34449.234161; stLENS3_333[644].fLow := 3.154572; stLENS3_333[644].fHigh := 7.943131;
    stLENS3_333[645].fEnergy := 34518.201574; stLENS3_333[645].fLow := 3.142123; stLENS3_333[645].fHigh := 7.909570;
    stLENS3_333[646].fEnergy := 34587.307059; stLENS3_333[646].fLow := 3.129723; stLENS3_333[646].fHigh := 7.876151;
    stLENS3_333[647].fEnergy := 34656.550894; stLENS3_333[647].fLow := 3.117372; stLENS3_333[647].fHigh := 7.842872;
    stLENS3_333[648].fEnergy := 34725.933355; stLENS3_333[648].fLow := 3.105070; stLENS3_333[648].fHigh := 7.809735;
    stLENS3_333[649].fEnergy := 34795.454720; stLENS3_333[649].fLow := 3.092816; stLENS3_333[649].fHigh := 7.776737;
    stLENS3_333[650].fEnergy := 34865.115267; stLENS3_333[650].fLow := 3.080610; stLENS3_333[650].fHigh := 7.743879;
    stLENS3_333[651].fEnergy := 34934.915274; stLENS3_333[651].fLow := 3.068453; stLENS3_333[651].fHigh := 7.711160;
    stLENS3_333[652].fEnergy := 35004.855021; stLENS3_333[652].fLow := 3.056344; stLENS3_333[652].fHigh := 7.678579;
    stLENS3_333[653].fEnergy := 35074.934788; stLENS3_333[653].fLow := 3.044282; stLENS3_333[653].fHigh := 7.646135;
    stLENS3_333[654].fEnergy := 35145.154854; stLENS3_333[654].fLow := 3.032268; stLENS3_333[654].fHigh := 7.613829;
    stLENS3_333[655].fEnergy := 35215.515501; stLENS3_333[655].fLow := 3.020302; stLENS3_333[655].fHigh := 7.581659;
    stLENS3_333[656].fEnergy := 35286.017010; stLENS3_333[656].fLow := 3.008383; stLENS3_333[656].fHigh := 7.549625;
    stLENS3_333[657].fEnergy := 35356.659663; stLENS3_333[657].fLow := 2.996510; stLENS3_333[657].fHigh := 7.517727;
    stLENS3_333[658].fEnergy := 35427.443743; stLENS3_333[658].fLow := 2.984685; stLENS3_333[658].fHigh := 7.485963;
    stLENS3_333[659].fEnergy := 35498.369532; stLENS3_333[659].fLow := 2.972906; stLENS3_333[659].fHigh := 7.454334;
    stLENS3_333[660].fEnergy := 35569.437315; stLENS3_333[660].fLow := 2.961174; stLENS3_333[660].fHigh := 7.422838;
    stLENS3_333[661].fEnergy := 35640.647376; stLENS3_333[661].fLow := 2.949488; stLENS3_333[661].fHigh := 7.391475;
    stLENS3_333[662].fEnergy := 35712.000000; stLENS3_333[662].fLow := 2.937848; stLENS3_333[662].fHigh := 7.360244;
    stLENS3_333[663].fEnergy := 35783.495472; stLENS3_333[663].fLow := 2.926254; stLENS3_333[663].fHigh := 7.329146;
    stLENS3_333[664].fEnergy := 35855.134077; stLENS3_333[664].fLow := 2.914706; stLENS3_333[664].fHigh := 7.298179;
    stLENS3_333[665].fEnergy := 35926.916104; stLENS3_333[665].fLow := 2.903204; stLENS3_333[665].fHigh := 7.267343;


